LIN {X 0,Y 135.979,Z 327.541,A -85,B 0,C 180,E1 -24797.792,E2 -24797.792} C_VEL
LIN {X 0,Y 136.06,Z 327.536,A -85,B 0,C 180,E1 -24801.701,E2 -24801.701} C_VEL
LIN {X 0,Y 136.276,Z 327.502,A -85,B 0,C 180,E1 -24805.604,E2 -24805.604} C_VEL
LIN {X 0,Y 136.39,Z 327.497,A -85,B 0,C 180,E1 -24808.988,E2 -24808.988} C_VEL
LIN {X 0,Y 135.911,Z 327.699,A -85,B 0,C 180,E1 -24810.982,E2 -24810.982} C_VEL
LIN {X 0,Y 135.083,Z 332.653,A -85,B 0,C 180,E1 -24817.037,E2 -24817.037} C_VEL
LIN {X 0,Y 134.416,Z 337.78,A -85,B 0,C 180,E1 -24823.292,E2 -24823.292} C_VEL
LIN {X 0,Y 135.153,Z 344.313,A -85,B 0,C 180,E1 -24831.118,E2 -24831.118} C_VEL
LIN {X 0,Y 135.675,Z 345.242,A -85,B 0,C 180,E1 -24832.189,E2 -24832.189} C_VEL
LIN {X 0,Y 136.863,Z 354.975,A -85,B 0,C 180,E1 -24833.739,E2 -24833.739} C_VEL
LIN {X 0,Y 136.657,Z 365.063,A -85,B 0,C 180,E1 -24835.949,E2 -24835.949} C_VEL
LIN {X 0,Y 136.414,Z 375.842,A -85,B 0,C 180,E1 -24838.897,E2 -24838.897} C_VEL
LIN {X 0,Y 136.178,Z 387.286,A -85,B 0,C 180,E1 -24842.962,E2 -24842.962} C_VEL
LIN {X 0,Y 136.68,Z 397.433,A -85,B 0,C 180,E1 -24847.389,E2 -24847.389} C_VEL
LIN {X 0,Y 138.168,Z 405.675,A -85,B 0,C 180,E1 -24851.743,E2 -24851.743} C_VEL
LIN {X 0,Y 140.736,Z 412.502,A -85,B 0,C 180,E1 -24855.945,E2 -24855.945} C_VEL
LIN {X 0,Y 144.351,Z 418.057,A -85,B 0,C 180,E1 -24859.93,E2 -24859.93} C_VEL
LIN {X 0,Y 148.855,Z 422.491,A -85,B 0,C 180,E1 -24863.664,E2 -24863.664} C_VEL
LIN {X 0,Y 154.201,Z 425.904,A -85,B 0,C 180,E1 -24867.118,E2 -24867.118} C_VEL
LIN {X 0,Y 158.207,Z 427.606,A -85,B 0,C 180,E1 -24869.255,E2 -24869.255} C_VEL
LIN {X 0,Y 162.506,Z 428.906,A -85,B 0,C 180,E1 -24871.267,E2 -24871.267} C_VEL
LIN {X 0,Y 170.287,Z 430.119,A -85,B 0,C 180,E1 -24874.368,E2 -24874.368} C_VEL
LIN {X 0,Y 176.196,Z 430.401,A -85,B 0,C 180,E1 -24876.752,E2 -24876.752} C_VEL
LIN {X 0,Y 178.308,Z 430.889,A -85,B 0,C 180,E1 -24879.1,E2 -24879.1} C_VEL
LIN {X 0,Y 179.822,Z 431.717,A -85,B 0,C 180,E1 -24882.048,E2 -24882.048} C_VEL
LIN {X 0,Y 179.602,Z 432.393,A -85,B 0,C 180,E1 -24883.62,E2 -24883.62} C_VEL
LIN {X 0,Y 177.592,Z 433.122,A -85,B 0,C 180,E1 -24884.575,E2 -24884.575} C_VEL
LIN {X 0,Y 167.705,Z 435.389,A -85,B 0,C 180,E1 -24887.893,E2 -24887.893} C_VEL
LIN {X 0,Y 158.877,Z 436.572,A -85,B 0,C 180,E1 -24891.735,E2 -24891.735} C_VEL
LIN {X 0,Y 151.362,Z 436.718,A -85,B 0,C 180,E1 -24896.139,E2 -24896.139} C_VEL
LIN {X 0,Y 145.311,Z 435.829,A -85,B 0,C 180,E1 -24901.076,E2 -24901.076} C_VEL
LIN {X 0,Y 141.019,Z 433.963,A -85,B 0,C 180,E1 -24906.503,E2 -24906.503} C_VEL
LIN {X 0,Y 138.563,Z 431.066,A -85,B 0,C 180,E1 -24912.282,E2 -24912.282} C_VEL
LIN {X 0,Y 138.068,Z 427.043,A -85,B 0,C 180,E1 -24918.252,E2 -24918.252} C_VEL
LIN {X 0,Y 139.403,Z 421.603,A -85,B 0,C 180,E1 -24924.213,E2 -24924.213} C_VEL
LIN {X 0,Y 140.672,Z 417.257,A -85,B 0,C 180,E1 -24927.791,E2 -24927.791} C_VEL
LIN {X 0,Y 142.352,Z 411.13,A -85,B 0,C 180,E1 -24931.702,E2 -24931.702} C_VEL
LIN {X 0,Y 144.37,Z 407.507,A -85,B 0,C 180,E1 -24933.874,E2 -24933.874} C_VEL
LIN {X 0,Y 141.887,Z 414.835,A -85,B 0,C 180,E1 -24937.82,E2 -24937.82} C_VEL
LIN {X 0,Y 140.373,Z 420.237,A -85,B 0,C 180,E1 -24941.553,E2 -24941.553} C_VEL
LIN {X 0,Y 139.886,Z 425.653,A -85,B 0,C 180,E1 -24946.414,E2 -24946.414} C_VEL
LIN {X 0,Y 141.433,Z 430.393,A -85,B 0,C 180,E1 -24951.881,E2 -24951.881} C_VEL
LIN {X 0,Y 144.15,Z 433.099,A -85,B 0,C 180,E1 -24956.027,E2 -24956.027} C_VEL
LIN {X 0,Y 146.64,Z 434.437,A -85,B 0,C 180,E1 -24958.638,E2 -24958.638} C_VEL
LIN {X 0,Y 149.609,Z 435.401,A -85,B 0,C 180,E1 -24961.114,E2 -24961.114} C_VEL
LIN {X 0,Y 153.036,Z 435.977,A -85,B 0,C 180,E1 -24963.442,E2 -24963.442} C_VEL
LIN {X 0,Y 156.96,Z 436.164,A -85,B 0,C 180,E1 -24965.598,E2 -24965.598} C_VEL
LIN {X 0,Y 161.236,Z 435.912,A -85,B 0,C 180,E1 -24967.607,E2 -24967.607} C_VEL
LIN {X 0,Y 165.846,Z 435.255,A -85,B 0,C 180,E1 -24969.468,E2 -24969.468} C_VEL
LIN {X 0,Y 170.838,Z 434.17,A -85,B 0,C 180,E1 -24971.164,E2 -24971.164} C_VEL
LIN {X 0,Y 178.821,Z 431.68,A -85,B 0,C 180,E1 -24973.455,E2 -24973.455} C_VEL
LIN {X 0,Y 183.487,Z 429.679,A -85,B 0,C 180,E1 -24974.829,E2 -24974.829} C_VEL
LIN {X 0,Y 182.659,Z 429.091,A -85,B 0,C 180,E1 -24976.974,E2 -24976.974} C_VEL
LIN {X 0,Y 181.359,Z 428.903,A -85,B 0,C 180,E1 -24978.79,E2 -24978.79} C_VEL
LIN {X 0,Y 178.916,Z 428.831,A -85,B 0,C 180,E1 -24981.058,E2 -24981.058} C_VEL
LIN {X 0,Y 176.005,Z 428.924,A -85,B 0,C 180,E1 -24983.201,E2 -24983.201} C_VEL
LIN {X 0,Y 172.17,Z 428.982,A -85,B 0,C 180,E1 -24985.143,E2 -24985.143} C_VEL
LIN {X 0,Y 167.361,Z 428.804,A -85,B 0,C 180,E1 -24986.91,E2 -24986.91} C_VEL
LIN {X 0,Y 162.753,Z 428.071,A -85,B 0,C 180,E1 -24988.786,E2 -24988.786} C_VEL
LIN {X 0,Y 158.415,Z 426.792,A -85,B 0,C 180,E1 -24990.787,E2 -24990.787} C_VEL
LIN {X 0,Y 152.538,Z 423.815,A -85,B 0,C 180,E1 -24994.039,E2 -24994.039} C_VEL
LIN {X 0,Y 150.428,Z 422.316,A -85,B 0,C 180,E1 -24995.385,E2 -24995.385} C_VEL
LIN {X 0,Y 147.381,Z 420.031,A -85,B 0,C 180,E1 -24997.089,E2 -24997.089} C_VEL
LIN {X 0,Y 143.823,Z 417.312,A -85,B 0,C 180,E1 -24998.608,E2 -24998.608} C_VEL
LIN {X 0,Y 137.001,Z 410.655,A -85,B 0,C 180,E1 -25001.573,E2 -25001.573} C_VEL
LIN {X 0,Y 134.667,Z 406.952,A -85,B 0,C 180,E1 -25003.278,E2 -25003.278} C_VEL
LIN {X 0,Y 134.183,Z 405.673,A -85,B 0,C 180,E1 -25003.906,E2 -25003.906} C_VEL
LIN {X 0,Y 132.351,Z 397.688,A -85,B 0,C 180,E1 -25007.733,E2 -25007.733} C_VEL
LIN {X 0,Y 131.623,Z 388.06,A -85,B 0,C 180,E1 -25011.552,E2 -25011.552} C_VEL
LIN {X 0,Y 131.713,Z 378.411,A -85,B 0,C 180,E1 -25014.638,E2 -25014.638} C_VEL
LIN {X 0,Y 132.18,Z 369.208,A -85,B 0,C 180,E1 -25016.948,E2 -25016.948} C_VEL
LIN {X 0,Y 132.386,Z 364.406,A -85,B 0,C 180,E1 -25017.904,E2 -25017.904} C_VEL
LIN {X 0,Y 127.928,Z 339.902,A -85,B 0,C 180,E1 -25036.759,E2 -25036.759} C_VEL
LIN {X 0,Y 128.249,Z 331.535,A -85,B 0,C 180,E1 -25043.405,E2 -25043.405} C_VEL
LIN {X 0,Y 128.472,Z 328.482,A -85,B 0,C 180,E1 -25045.948,E2 -25045.948} C_VEL
LIN {X 0,Y 128.911,Z 328.428,A -85,B 0,C 180,E1 -25049.379,E2 -25049.379} C_VEL
LIN {X 0,Y 128.987,Z 328.412,A -85,B 0,C 180,E1 -25055.185,E2 -25055.185} C_VEL
LIN {X 0,Y 128.917,Z 328.425,A -85,B 0,C 180,E1 -25060.852,E2 -25060.852} C_VEL
LIN {X 0,Y 128.905,Z 328.426,A -85,B 0,C 180,E1 -25065.129,E2 -25065.129} C_VEL
LIN {X 0,Y 128.928,Z 328.422,A -85,B 0,C 180,E1 -25069.736,E2 -25069.736} C_VEL
LIN {X 0,Y 128.973,Z 328.42,A -85,B 0,C 180,E1 -25074.816,E2 -25074.816} C_VEL
LIN {X 0,Y 129.008,Z 328.409,A -85,B 0,C 180,E1 -25080.64,E2 -25080.64} C_VEL
LIN {X 0,Y 129.022,Z 328.413,A -85,B 0,C 180,E1 -25084.166,E2 -25084.166} C_VEL
LIN {X 0,Y 129.099,Z 328.399,A -85,B 0,C 180,E1 -25087.726,E2 -25087.726} C_VEL
LIN {X 0,Y 129.147,Z 328.397,A -85,B 0,C 180,E1 -25090.943,E2 -25090.943} C_VEL
LIN {X 0,Y 129.38,Z 328.362,A -85,B 0,C 180,E1 -25097.875,E2 -25097.875} C_VEL
LIN {X 0,Y 129.461,Z 328.359,A -85,B 0,C 180,E1 -25100.627,E2 -25100.627} C_VEL
LIN {X 0,Y 130.057,Z 328.286,A -85,B 0,C 180,E1 -25110,E2 -25110} C_VEL
LIN {X 0,Y 129.461,Z 328.359,A -85,B 0,C 180,E1 -25119.373,E2 -25119.373} C_VEL
LIN {X 0,Y 129.336,Z 328.367,A -85,B 0,C 180,E1 -25122.554,E2 -25122.554} C_VEL
LIN {X 0,Y 129.17,Z 328.394,A -85,B 0,C 180,E1 -25129.054,E2 -25129.054} C_VEL
LIN {X 0,Y 129.127,Z 328.396,A -85,B 0,C 180,E1 -25132.395,E2 -25132.395} C_VEL
LIN {X 0,Y 129.028,Z 328.407,A -85,B 0,C 180,E1 -25139.376,E2 -25139.376} C_VEL
LIN {X 0,Y 128.973,Z 328.42,A -85,B 0,C 180,E1 -25145.184,E2 -25145.184} C_VEL
LIN {X 0,Y 128.917,Z 328.424,A -85,B 0,C 180,E1 -25150.858,E2 -25150.858} C_VEL
LIN {X 0,Y 128.905,Z 328.425,A -85,B 0,C 180,E1 -25155.135,E2 -25155.135} C_VEL
LIN {X 0,Y 128.942,Z 328.422,A -85,B 0,C 180,E1 -25159.736,E2 -25159.736} C_VEL
LIN {X 0,Y 129.139,Z 328.394,A -85,B 0,C 180,E1 -25164.72,E2 -25164.72} C_VEL
LIN {X 0,Y 129.235,Z 328.383,A -85,B 0,C 180,E1 -25167.061,E2 -25167.061} C_VEL
LIN {X 0,Y 128.692,Z 328.577,A -85,B 0,C 180,E1 -25171.572,E2 -25171.572} C_VEL
LIN {X 0,Y 127.933,Z 333.105,A -85,B 0,C 180,E1 -25177.389,E2 -25177.389} C_VEL
LIN {X 0,Y 127.276,Z 338.27,A -85,B 0,C 180,E1 -25183.977,E2 -25183.977} C_VEL
LIN {X 0,Y 128.495,Z 344.938,A -85,B 0,C 180,E1 -25192.351,E2 -25192.351} C_VEL
LIN {X 0,Y 128.938,Z 345.731,A -85,B 0,C 180,E1 -25193.148,E2 -25193.148} C_VEL
LIN {X 0,Y 130.047,Z 354.44,A -85,B 0,C 180,E1 -25194.577,E2 -25194.577} C_VEL
LIN {X 0,Y 129.881,Z 364.497,A -85,B 0,C 180,E1 -25196.902,E2 -25196.902} C_VEL
LIN {X 0,Y 129.768,Z 374.013,A -85,B 0,C 180,E1 -25199.616,E2 -25199.616} C_VEL
LIN {X 0,Y 129.529,Z 383.947,A -85,B 0,C 180,E1 -25203.114,E2 -25203.114} C_VEL
LIN {X 0,Y 129.858,Z 393.128,A -85,B 0,C 180,E1 -25206.998,E2 -25206.998} C_VEL
LIN {X 0,Y 131.157,Z 402.14,A -85,B 0,C 180,E1 -25211.596,E2 -25211.596} C_VEL
LIN {X 0,Y 133.538,Z 409.687,A -85,B 0,C 180,E1 -25216.044,E2 -25216.044} C_VEL
LIN {X 0,Y 137.758,Z 416.78,A -85,B 0,C 180,E1 -25220.927,E2 -25220.927} C_VEL
LIN {X 0,Y 142.391,Z 421.671,A -85,B 0,C 180,E1 -25224.809,E2 -25224.809} C_VEL
LIN {X 0,Y 147.893,Z 425.491,A -85,B 0,C 180,E1 -25228.377,E2 -25228.377} C_VEL
LIN {X 0,Y 152.021,Z 427.502,A -85,B 0,C 180,E1 -25230.57,E2 -25230.57} C_VEL
LIN {X 0,Y 156.454,Z 429.083,A -85,B 0,C 180,E1 -25232.622,E2 -25232.622} C_VEL
LIN {X 0,Y 164.94,Z 430.874,A -85,B 0,C 180,E1 -25235.945,E2 -25235.945} C_VEL
LIN {X 0,Y 166.079,Z 431.002,A -85,B 0,C 180,E1 -25236.334,E2 -25236.334} C_VEL
LIN {X 0,Y 170.321,Z 431.518,A -85,B 0,C 180,E1 -25238.243,E2 -25238.243} C_VEL
LIN {X 0,Y 172.095,Z 432.303,A -85,B 0,C 180,E1 -25240.802,E2 -25240.802} C_VEL
LIN {X 0,Y 172.594,Z 433.048,A -85,B 0,C 180,E1 -25242.865,E2 -25242.865} C_VEL
LIN {X 0,Y 162.533,Z 434.785,A -85,B 0,C 180,E1 -25246.223,E2 -25246.223} C_VEL
LIN {X 0,Y 153.433,Z 435.466,A -85,B 0,C 180,E1 -25250.113,E2 -25250.113} C_VEL
LIN {X 0,Y 145.65,Z 435.17,A -85,B 0,C 180,E1 -25254.617,E2 -25254.617} C_VEL
LIN {X 0,Y 139.369,Z 433.885,A -85,B 0,C 180,E1 -25259.717,E2 -25259.717} C_VEL
LIN {X 0,Y 134.86,Z 431.648,A -85,B 0,C 180,E1 -25265.36,E2 -25265.36} C_VEL
LIN {X 0,Y 132.281,Z 428.393,A -85,B 0,C 180,E1 -25271.411,E2 -25271.411} C_VEL
LIN {X 0,Y 131.754,Z 424.034,A -85,B 0,C 180,E1 -25277.68,E2 -25277.68} C_VEL
LIN {X 0,Y 133.18,Z 418.274,A -85,B 0,C 180,E1 -25283.942,E2 -25283.942} C_VEL
LIN {X 0,Y 134.503,Z 413.642,A -85,B 0,C 180,E1 -25287.69,E2 -25287.69} C_VEL
LIN {X 0,Y 136.475,Z 406.993,A -85,B 0,C 180,E1 -25291.898,E2 -25291.898} C_VEL
LIN {X 0,Y 138.897,Z 403.116,A -85,B 0,C 180,E1 -25294.28,E2 -25294.28} C_VEL
LIN {X 0,Y 136.176,Z 410.644,A -85,B 0,C 180,E1 -25298.15,E2 -25298.15} C_VEL
LIN {X 0,Y 134.564,Z 416.341,A -85,B 0,C 180,E1 -25302.059,E2 -25302.059} C_VEL
LIN {X 0,Y 133.906,Z 421.325,A -85,B 0,C 180,E1 -25306.284,E2 -25306.284} C_VEL
LIN {X 0,Y 134.814,Z 426.291,A -85,B 0,C 180,E1 -25311.403,E2 -25311.403} C_VEL
LIN {X 0,Y 136.199,Z 428.656,A -85,B 0,C 180,E1 -25314.381,E2 -25314.381} C_VEL
LIN {X 0,Y 138.201,Z 430.639,A -85,B 0,C 180,E1 -25317.238,E2 -25317.238} C_VEL
LIN {X 0,Y 140.76,Z 432.23,A -85,B 0,C 180,E1 -25319.953,E2 -25319.953} C_VEL
LIN {X 0,Y 147.323,Z 434.326,A -85,B 0,C 180,E1 -25324.922,E2 -25324.922} C_VEL
LIN {X 0,Y 151.341,Z 434.852,A -85,B 0,C 180,E1 -25327.135,E2 -25327.135} C_VEL
LIN {X 0,Y 155.732,Z 434.988,A -85,B 0,C 180,E1 -25329.184,E2 -25329.184} C_VEL
LIN {X 0,Y 160.443,Z 434.685,A -85,B 0,C 180,E1 -25331.076,E2 -25331.076} C_VEL
LIN {X 0,Y 165.554,Z 433.973,A -85,B 0,C 180,E1 -25332.783,E2 -25332.783} C_VEL
LIN {X 0,Y 170.948,Z 432.822,A -85,B 0,C 180,E1 -25334.339,E2 -25334.339} C_VEL
LIN {X 0,Y 176.254,Z 431.265,A -85,B 0,C 180,E1 -25335.868,E2 -25335.868} C_VEL
LIN {X 0,Y 175.546,Z 430.96,A -85,B 0,C 180,E1 -25337.106,E2 -25337.106} C_VEL
LIN {X 0,Y 173.23,Z 430.557,A -85,B 0,C 180,E1 -25339.521,E2 -25339.521} C_VEL
LIN {X 0,Y 170.342,Z 430.266,A -85,B 0,C 180,E1 -25341.763,E2 -25341.763} C_VEL
LIN {X 0,Y 166.388,Z 429.931,A -85,B 0,C 180,E1 -25343.744,E2 -25343.744} C_VEL
LIN {X 0,Y 161.432,Z 429.339,A -85,B 0,C 180,E1 -25345.527,E2 -25345.527} C_VEL
LIN {X 0,Y 156.681,Z 428.21,A -85,B 0,C 180,E1 -25347.431,E2 -25347.431} C_VEL
LIN {X 0,Y 150.121,Z 425.546,A -85,B 0,C 180,E1 -25350.553,E2 -25350.553} C_VEL
LIN {X 0,Y 144.328,Z 421.541,A -85,B 0,C 180,E1 -25354.004,E2 -25354.004} C_VEL
LIN {X 0,Y 139.447,Z 416.299,A -85,B 0,C 180,E1 -25357.787,E2 -25357.787} C_VEL
LIN {X 0,Y 136.156,Z 410.722,A -85,B 0,C 180,E1 -25361.175,E2 -25361.175} C_VEL
LIN {X 0,Y 134.183,Z 405.673,A -85,B 0,C 180,E1 -25363.906,E2 -25363.906} C_VEL
LIN {X 0,Y 132.597,Z 401.763,A -85,B 0,C 180,E1 -25365.657,E2 -25365.657} C_VEL
LIN {X 0,Y 129.033,Z 394.378,A -85,B 0,C 180,E1 -25368.074,E2 -25368.074} C_VEL
LIN {X 0,Y 126.08,Z 386.22,A -85,B 0,C 180,E1 -25370.333,E2 -25370.333} C_VEL
LIN {X 0,Y 125.532,Z 381.233,A -85,B 0,C 180,E1 -25371.814,E2 -25371.814} C_VEL
LIN {X 0,Y 125.79,Z 372.273,A -85,B 0,C 180,E1 -25374.385,E2 -25374.385} C_VEL
LIN {X 0,Y 126.176,Z 365.058,A -85,B 0,C 180,E1 -25376.103,E2 -25376.103} C_VEL
LIN {X 0,Y 120.807,Z 340.148,A -85,B 0,C 180,E1 -25396.037,E2 -25396.037} C_VEL
LIN {X 0,Y 121.1,Z 332.348,A -85,B 0,C 180,E1 -25402.529,E2 -25402.529} C_VEL
LIN {X 0,Y 121.308,Z 329.374,A -85,B 0,C 180,E1 -25405.06,E2 -25405.06} C_VEL
LIN {X 0,Y 121.862,Z 329.305,A -85,B 0,C 180,E1 -25410.108,E2 -25410.108} C_VEL
LIN {X 0,Y 121.899,Z 329.298,A -85,B 0,C 180,E1 -25416.18,E2 -25416.18} C_VEL
LIN {X 0,Y 121.857,Z 329.301,A -85,B 0,C 180,E1 -25421.43,E2 -25421.43} C_VEL
LIN {X 0,Y 121.857,Z 329.306,A -85,B 0,C 180,E1 -25428.563,E2 -25428.563} C_VEL
LIN {X 0,Y 121.925,Z 329.298,A -85,B 0,C 180,E1 -25434.801,E2 -25434.801} C_VEL
LIN {X 0,Y 121.92,Z 329.291,A -85,B 0,C 180,E1 -25439.834,E2 -25439.834} C_VEL
LIN {X 0,Y 121.975,Z 329.29,A -85,B 0,C 180,E1 -25446.213,E2 -25446.213} C_VEL
LIN {X 0,Y 122.038,Z 329.278,A -85,B 0,C 180,E1 -25449.786,E2 -25449.786} C_VEL
LIN {X 0,Y 122.231,Z 329.252,A -85,B 0,C 180,E1 -25456.703,E2 -25456.703} C_VEL
LIN {X 0,Y 122.398,Z 329.238,A -85,B 0,C 180,E1 -25460.081,E2 -25460.081} C_VEL
LIN {X 0,Y 122.551,Z 329.215,A -85,B 0,C 180,E1 -25466.712,E2 -25466.712} C_VEL
LIN {X 0,Y 123.011,Z 329.163,A -85,B 0,C 180,E1 -25470,E2 -25470} C_VEL
LIN {X 0,Y 122.4,Z 329.237,A -85,B 0,C 180,E1 -25476.594,E2 -25476.594} C_VEL
LIN {X 0,Y 122.398,Z 329.238,A -85,B 0,C 180,E1 -25479.919,E2 -25479.919} C_VEL
LIN {X 0,Y 122.232,Z 329.252,A -85,B 0,C 180,E1 -25483.296,E2 -25483.296} C_VEL
LIN {X 0,Y 122.06,Z 329.276,A -85,B 0,C 180,E1 -25490.211,E2 -25490.211} C_VEL
LIN {X 0,Y 121.988,Z 329.289,A -85,B 0,C 180,E1 -25493.784,E2 -25493.784} C_VEL
LIN {X 0,Y 121.933,Z 329.289,A -85,B 0,C 180,E1 -25500.176,E2 -25500.176} C_VEL
LIN {X 0,Y 121.889,Z 329.3,A -85,B 0,C 180,E1 -25506.183,E2 -25506.183} C_VEL
LIN {X 0,Y 121.857,Z 329.306,A -85,B 0,C 180,E1 -25511.437,E2 -25511.437} C_VEL
LIN {X 0,Y 121.864,Z 329.3,A -85,B 0,C 180,E1 -25518.566,E2 -25518.566} C_VEL
LIN {X 0,Y 122.094,Z 329.27,A -85,B 0,C 180,E1 -25524.862,E2 -25524.862} C_VEL
LIN {X 0,Y 121.889,Z 329.304,A -85,B 0,C 180,E1 -25529.87,E2 -25529.87} C_VEL
LIN {X 0,Y 121.452,Z 329.586,A -85,B 0,C 180,E1 -25532.429,E2 -25532.429} C_VEL
LIN {X 0,Y 120.678,Z 334.258,A -85,B 0,C 180,E1 -25538.718,E2 -25538.718} C_VEL
LIN {X 0,Y 120.883,Z 343.579,A -85,B 0,C 180,E1 -25551.251,E2 -25551.251} C_VEL
LIN {X 0,Y 122.276,Z 345.925,A -85,B 0,C 180,E1 -25554.232,E2 -25554.232} C_VEL
LIN {X 0,Y 123.425,Z 355.351,A -85,B 0,C 180,E1 -25555.923,E2 -25555.923} C_VEL
LIN {X 0,Y 123.225,Z 368.066,A -85,B 0,C 180,E1 -25559.187,E2 -25559.187} C_VEL
LIN {X 0,Y 122.989,Z 378.06,A -85,B 0,C 180,E1 -25562.461,E2 -25562.461} C_VEL
LIN {X 0,Y 123.176,Z 388.165,A -85,B 0,C 180,E1 -25566.557,E2 -25566.557} C_VEL
LIN {X 0,Y 124.25,Z 398.142,A -85,B 0,C 180,E1 -25571.423,E2 -25571.423} C_VEL
LIN {X 0,Y 126.499,Z 406.389,A -85,B 0,C 180,E1 -25576.132,E2 -25576.132} C_VEL
LIN {X 0,Y 130.564,Z 414.29,A -85,B 0,C 180,E1 -25581.309,E2 -25581.309} C_VEL
LIN {X 0,Y 134.328,Z 418.931,A -85,B 0,C 180,E1 -25584.747,E2 -25584.747} C_VEL
LIN {X 0,Y 139.699,Z 423.542,A -85,B 0,C 180,E1 -25588.554,E2 -25588.554} C_VEL
LIN {X 0,Y 145.932,Z 427.144,A -85,B 0,C 180,E1 -25591.993,E2 -25591.993} C_VEL
LIN {X 0,Y 155.328,Z 430.504,A -85,B 0,C 180,E1 -25596.033,E2 -25596.033} C_VEL
LIN {X 0,Y 160.37,Z 431.552,A -85,B 0,C 180,E1 -25597.849,E2 -25597.849} C_VEL
LIN {X 0,Y 163.896,Z 432.229,A -85,B 0,C 180,E1 -25599.479,E2 -25599.479} C_VEL
LIN {X 0,Y 165.011,Z 433.181,A -85,B 0,C 180,E1 -25601.975,E2 -25601.975} C_VEL
LIN {X 0,Y 157.538,Z 433.935,A -85,B 0,C 180,E1 -25604.456,E2 -25604.456} C_VEL
LIN {X 0,Y 148.162,Z 434.139,A -85,B 0,C 180,E1 -25608.388,E2 -25608.388} C_VEL
LIN {X 0,Y 140.086,Z 433.385,A -85,B 0,C 180,E1 -25612.984,E2 -25612.984} C_VEL
LIN {X 0,Y 133.563,Z 431.721,A -85,B 0,C 180,E1 -25618.251,E2 -25618.251} C_VEL
LIN {X 0,Y 128.849,Z 429.116,A -85,B 0,C 180,E1 -25624.128,E2 -25624.128} C_VEL
LIN {X 0,Y 125.85,Z 424.735,A -85,B 0,C 180,E1 -25631.698,E2 -25631.698} C_VEL
LIN {X 0,Y 125.791,Z 419.455,A -85,B 0,C 180,E1 -25638.723,E2 -25638.723} C_VEL
LIN {X 0,Y 127.211,Z 414.357,A -85,B 0,C 180,E1 -25643.992,E2 -25643.992} C_VEL
LIN {X 0,Y 128.499,Z 409.542,A -85,B 0,C 180,E1 -25647.757,E2 -25647.757} C_VEL
LIN {X 0,Y 130.924,Z 402.291,A -85,B 0,C 180,E1 -25652.307,E2 -25652.307} C_VEL
LIN {X 0,Y 133.56,Z 398.564,A -85,B 0,C 180,E1 -25654.716,E2 -25654.716} C_VEL
LIN {X 0,Y 130.81,Z 405.888,A -85,B 0,C 180,E1 -25658.416,E2 -25658.416} C_VEL
LIN {X 0,Y 128.929,Z 412.216,A -85,B 0,C 180,E1 -25662.594,E2 -25662.594} C_VEL
LIN {X 0,Y 128.158,Z 418.801,A -85,B 0,C 180,E1 -25668.165,E2 -25668.165} C_VEL
LIN {X 0,Y 129.01,Z 422.93,A -85,B 0,C 180,E1 -25672.417,E2 -25672.417} C_VEL
LIN {X 0,Y 131.341,Z 426.786,A -85,B 0,C 180,E1 -25677.054,E2 -25677.054} C_VEL
LIN {X 0,Y 135.044,Z 429.761,A -85,B 0,C 180,E1 -25681.361,E2 -25681.361} C_VEL
LIN {X 0,Y 138.185,Z 431.276,A -85,B 0,C 180,E1 -25684.018,E2 -25684.018} C_VEL
LIN {X 0,Y 141.777,Z 432.39,A -85,B 0,C 180,E1 -25686.502,E2 -25686.502} C_VEL
LIN {X 0,Y 145.893,Z 433.221,A -85,B 0,C 180,E1 -25688.773,E2 -25688.773} C_VEL
LIN {X 0,Y 150.387,Z 433.687,A -85,B 0,C 180,E1 -25690.864,E2 -25690.864} C_VEL
LIN {X 0,Y 155.207,Z 433.782,A -85,B 0,C 180,E1 -25692.783,E2 -25692.783} C_VEL
LIN {X 0,Y 160.428,Z 433.469,A -85,B 0,C 180,E1 -25694.502,E2 -25694.502} C_VEL
LIN {X 0,Y 167.727,Z 432.402,A -85,B 0,C 180,E1 -25696.565,E2 -25696.565} C_VEL
LIN {X 0,Y 167.485,Z 431.957,A -85,B 0,C 180,E1 -25697.822,E2 -25697.822} C_VEL
LIN {X 0,Y 164.707,Z 431.269,A -85,B 0,C 180,E1 -25700.201,E2 -25700.201} C_VEL
LIN {X 0,Y 160.685,Z 430.594,A -85,B 0,C 180,E1 -25702.238,E2 -25702.238} C_VEL
LIN {X 0,Y 155.588,Z 429.599,A -85,B 0,C 180,E1 -25704.036,E2 -25704.036} C_VEL
LIN {X 0,Y 148.408,Z 427.12,A -85,B 0,C 180,E1 -25706.999,E2 -25706.999} C_VEL
LIN {X 0,Y 141.923,Z 423.402,A -85,B 0,C 180,E1 -25710.313,E2 -25710.313} C_VEL
LIN {X 0,Y 136.297,Z 418.421,A -85,B 0,C 180,E1 -25714.001,E2 -25714.001} C_VEL
LIN {X 0,Y 131.672,Z 411.986,A -85,B 0,C 180,E1 -25718.057,E2 -25718.057} C_VEL
LIN {X 0,Y 128.127,Z 403.878,A -85,B 0,C 180,E1 -25722.504,E2 -25722.504} C_VEL
LIN {X 0,Y 126.334,Z 395.716,A -85,B 0,C 180,E1 -25726.32,E2 -25726.32} C_VEL
LIN {X 0,Y 125.556,Z 386.77,A -85,B 0,C 180,E1 -25729.922,E2 -25729.922} C_VEL
LIN {X 0,Y 125.532,Z 381.233,A -85,B 0,C 180,E1 -25731.814,E2 -25731.814} C_VEL
LIN {X 0,Y 124.969,Z 377.479,A -85,B 0,C 180,E1 -25732.765,E2 -25732.765} C_VEL
LIN {X 0,Y 123.008,Z 371.864,A -85,B 0,C 180,E1 -25733.566,E2 -25733.566} C_VEL
LIN {X 0,Y 120.22,Z 365.879,A -85,B 0,C 180,E1 -25734.727,E2 -25734.727} C_VEL
LIN {X 0,Y 119.024,Z 363.495,A -85,B 0,C 180,E1 -25735.761,E2 -25735.761} C_VEL
LIN {X 0,Y 118.831,Z 363.119,A -85,B 0,C 180,E1 -25736.022,E2 -25736.022} C_VEL
LIN {X 0,Y 113.76,Z 339.277,A -85,B 0,C 180,E1 -25756.136,E2 -25756.136} C_VEL
LIN {X 0,Y 114.025,Z 332.111,A -85,B 0,C 180,E1 -25762.402,E2 -25762.402} C_VEL
LIN {X 0,Y 114.122,Z 330.268,A -85,B 0,C 180,E1 -25764.19,E2 -25764.19} C_VEL
LIN {X 0,Y 114.702,Z 330.198,A -85,B 0,C 180,E1 -25769.346,E2 -25769.346} C_VEL
LIN {X 0,Y 114.818,Z 330.176,A -85,B 0,C 180,E1 -25773.422,E2 -25773.422} C_VEL
LIN {X 0,Y 114.783,Z 330.187,A -85,B 0,C 180,E1 -25777.749,E2 -25777.749} C_VEL
LIN {X 0,Y 114.771,Z 330.182,A -85,B 0,C 180,E1 -25782.708,E2 -25782.708} C_VEL
LIN {X 0,Y 114.779,Z 330.187,A -85,B 0,C 180,E1 -25787.659,E2 -25787.659} C_VEL
LIN {X 0,Y 114.788,Z 330.181,A -85,B 0,C 180,E1 -25792.736,E2 -25792.736} C_VEL
LIN {X 0,Y 114.854,Z 330.172,A -85,B 0,C 180,E1 -25798.935,E2 -25798.935} C_VEL
LIN {X 0,Y 114.939,Z 330.165,A -85,B 0,C 180,E1 -25806.504,E2 -25806.504} C_VEL
LIN {X 0,Y 115.004,Z 330.16,A -85,B 0,C 180,E1 -25812.208,E2 -25812.208} C_VEL
LIN {X 0,Y 115.239,Z 330.122,A -85,B 0,C 180,E1 -25817.34,E2 -25817.34} C_VEL
LIN {X 0,Y 115.344,Z 330.116,A -85,B 0,C 180,E1 -25823,E2 -25823} C_VEL
LIN {X 0,Y 115.963,Z 330.041,A -85,B 0,C 180,E1 -25830,E2 -25830} C_VEL
LIN {X 0,Y 115.344,Z 330.116,A -85,B 0,C 180,E1 -25837,E2 -25837} C_VEL
LIN {X 0,Y 115.239,Z 330.122,A -85,B 0,C 180,E1 -25842.66,E2 -25842.66} C_VEL
LIN {X 0,Y 115.017,Z 330.158,A -85,B 0,C 180,E1 -25847.79,E2 -25847.79} C_VEL
LIN {X 0,Y 114.957,Z 330.163,A -85,B 0,C 180,E1 -25853.516,E2 -25853.516} C_VEL
LIN {X 0,Y 114.859,Z 330.172,A -85,B 0,C 180,E1 -25861.07,E2 -25861.07} C_VEL
LIN {X 0,Y 114.777,Z 330.181,A -85,B 0,C 180,E1 -25867.757,E2 -25867.757} C_VEL
LIN {X 0,Y 114.772,Z 330.189,A -85,B 0,C 180,E1 -25872.716,E2 -25872.716} C_VEL
LIN {X 0,Y 114.784,Z 330.181,A -85,B 0,C 180,E1 -25877.668,E2 -25877.668} C_VEL
LIN {X 0,Y 114.901,Z 330.172,A -85,B 0,C 180,E1 -25882.67,E2 -25882.67} C_VEL
LIN {X 0,Y 114.904,Z 330.172,A -85,B 0,C 180,E1 -25888.904,E2 -25888.904} C_VEL
LIN {X 0,Y 114.257,Z 330.334,A -85,B 0,C 180,E1 -25893.028,E2 -25893.028} C_VEL
LIN {X 0,Y 113.639,Z 333.95,A -85,B 0,C 180,E1 -25898.224,E2 -25898.224} C_VEL
LIN {X 0,Y 114.327,Z 344.329,A -85,B 0,C 180,E1 -25912.943,E2 -25912.943} C_VEL
LIN {X 0,Y 115.715,Z 346.303,A -85,B 0,C 180,E1 -25915.541,E2 -25915.541} C_VEL
LIN {X 0,Y 116.761,Z 354.204,A -85,B 0,C 180,E1 -25916.986,E2 -25916.986} C_VEL
LIN {X 0,Y 116.654,Z 365.828,A -85,B 0,C 180,E1 -25920.004,E2 -25920.004} C_VEL
LIN {X 0,Y 116.537,Z 376.02,A -85,B 0,C 180,E1 -25923.462,E2 -25923.462} C_VEL
LIN {X 0,Y 116.792,Z 386.477,A -85,B 0,C 180,E1 -25927.786,E2 -25927.786} C_VEL
LIN {X 0,Y 117.714,Z 395.232,A -85,B 0,C 180,E1 -25932.066,E2 -25932.066} C_VEL
LIN {X 0,Y 120.466,Z 405.263,A -85,B 0,C 180,E1 -25937.84,E2 -25937.84} C_VEL
LIN {X 0,Y 124.129,Z 412.417,A -85,B 0,C 180,E1 -25942.473,E2 -25942.473} C_VEL
LIN {X 0,Y 129.751,Z 419.22,A -85,B 0,C 180,E1 -25947.417,E2 -25947.417} C_VEL
LIN {X 0,Y 135.559,Z 423.932,A -85,B 0,C 180,E1 -25951.232,E2 -25951.232} C_VEL
LIN {X 0,Y 142.252,Z 427.678,A -85,B 0,C 180,E1 -25954.626,E2 -25954.626} C_VEL
LIN {X 0,Y 149.592,Z 430.489,A -85,B 0,C 180,E1 -25957.648,E2 -25957.648} C_VEL
LIN {X 0,Y 154.781,Z 431.839,A -85,B 0,C 180,E1 -25959.475,E2 -25959.475} C_VEL
LIN {X 0,Y 156.919,Z 432.398,A -85,B 0,C 180,E1 -25960.413,E2 -25960.413} C_VEL
LIN {X 0,Y 152.722,Z 432.835,A -85,B 0,C 180,E1 -25962.583,E2 -25962.583} C_VEL
LIN {X 0,Y 143.06,Z 432.552,A -85,B 0,C 180,E1 -25966.546,E2 -25966.546} C_VEL
LIN {X 0,Y 134.717,Z 431.364,A -85,B 0,C 180,E1 -25971.242,E2 -25971.242} C_VEL
LIN {X 0,Y 127.912,Z 429.319,A -85,B 0,C 180,E1 -25976.671,E2 -25976.671} C_VEL
LIN {X 0,Y 122.976,Z 426.351,A -85,B 0,C 180,E1 -25982.794,E2 -25982.794} C_VEL
LIN {X 0,Y 119.812,Z 421.584,A -85,B 0,C 180,E1 -25990.74,E2 -25990.74} C_VEL
LIN {X 0,Y 119.763,Z 415.948,A -85,B 0,C 180,E1 -25998.148,E2 -25998.148} C_VEL
LIN {X 0,Y 121.113,Z 410.949,A -85,B 0,C 180,E1 -26003.335,E2 -26003.335} C_VEL
LIN {X 0,Y 122.277,Z 406.806,A -85,B 0,C 180,E1 -26006.705,E2 -26006.705} C_VEL
LIN {X 0,Y 124.634,Z 399.195,A -85,B 0,C 180,E1 -26011.616,E2 -26011.616} C_VEL
LIN {X 0,Y 126.796,Z 395.558,A -85,B 0,C 180,E1 -26013.835,E2 -26013.835} C_VEL
LIN {X 0,Y 128.536,Z 393.657,A -85,B 0,C 180,E1 -26015.127,E2 -26015.127} C_VEL
LIN {X 0,Y 125.098,Z 402.518,A -85,B 0,C 180,E1 -26019.703,E2 -26019.703} C_VEL
LIN {X 0,Y 123.205,Z 409.041,A -85,B 0,C 180,E1 -26024.117,E2 -26024.117} C_VEL
LIN {X 0,Y 122.567,Z 414.17,A -85,B 0,C 180,E1 -26028.383,E2 -26028.383} C_VEL
LIN {X 0,Y 123.787,Z 420.483,A -85,B 0,C 180,E1 -26034.706,E2 -26034.706} C_VEL
LIN {X 0,Y 126.859,Z 424.771,A -85,B 0,C 180,E1 -26039.908,E2 -26039.908} C_VEL
LIN {X 0,Y 129.517,Z 426.962,A -85,B 0,C 180,E1 -26042.863,E2 -26042.863} C_VEL
LIN {X 0,Y 132.745,Z 428.771,A -85,B 0,C 180,E1 -26045.618,E2 -26045.618} C_VEL
LIN {X 0,Y 136.426,Z 430.215,A -85,B 0,C 180,E1 -26048.184,E2 -26048.184} C_VEL
LIN {X 0,Y 145.229,Z 432.072,A -85,B 0,C 180,E1 -26052.649,E2 -26052.649} C_VEL
LIN {X 0,Y 150.156,Z 432.496,A -85,B 0,C 180,E1 -26054.594,E2 -26054.594} C_VEL
LIN {X 0,Y 159.42,Z 432.357,A -85,B 0,C 180,E1 -26057.433,E2 -26057.433} C_VEL
LIN {X 0,Y 159.032,Z 431.957,A -85,B 0,C 180,E1 -26058.476,E2 -26058.476} C_VEL
LIN {X 0,Y 158.608,Z 431.793,A -85,B 0,C 180,E1 -26058.875,E2 -26058.875} C_VEL
LIN {X 0,Y 155.088,Z 430.954,A -85,B 0,C 180,E1 -26060.619,E2 -26060.619} C_VEL
LIN {X 0,Y 149.845,Z 429.555,A -85,B 0,C 180,E1 -26062.427,E2 -26062.427} C_VEL
LIN {X 0,Y 142.49,Z 426.401,A -85,B 0,C 180,E1 -26065.44,E2 -26065.44} C_VEL
LIN {X 0,Y 135.828,Z 422.14,A -85,B 0,C 180,E1 -26068.837,E2 -26068.837} C_VEL
LIN {X 0,Y 130.1,Z 416.449,A -85,B 0,C 180,E1 -26072.662,E2 -26072.662} C_VEL
LIN {X 0,Y 125.416,Z 409.436,A -85,B 0,C 180,E1 -26076.9,E2 -26076.9} C_VEL
LIN {X 0,Y 121.922,Z 400.605,A -85,B 0,C 180,E1 -26081.512,E2 -26081.512} C_VEL
LIN {X 0,Y 120.474,Z 393.561,A -85,B 0,C 180,E1 -26084.776,E2 -26084.776} C_VEL
LIN {X 0,Y 119.672,Z 384.05,A -85,B 0,C 180,E1 -26088.564,E2 -26088.564} C_VEL
LIN {X 0,Y 119.742,Z 373.448,A -85,B 0,C 180,E1 -26091.983,E2 -26091.983} C_VEL
LIN {X 0,Y 120.131,Z 365.866,A -85,B 0,C 180,E1 -26093.909,E2 -26093.909} C_VEL
LIN {X 0,Y 118.831,Z 363.119,A -85,B 0,C 180,E1 -26096.022,E2 -26096.022} C_VEL
LIN {X 0,Y 116.786,Z 360.054,A -85,B 0,C 180,E1 -26098.27,E2 -26098.27} C_VEL
LIN {X 0,Y 108.203,Z 349.832,A -85,B 0,C 180,E1 -26105.754,E2 -26105.754} C_VEL
LIN {X 0,Y 107.036,Z 346.797,A -85,B 0,C 180,E1 -26108.383,E2 -26108.383} C_VEL
LIN {X 0,Y 106.787,Z 336.183,A -85,B 0,C 180,E1 -26118.211,E2 -26118.211} C_VEL
LIN {X 0,Y 106.979,Z 331.16,A -85,B 0,C 180,E1 -26122.963,E2 -26122.963} C_VEL
LIN {X 0,Y 107.387,Z 331.109,A -85,B 0,C 180,E1 -26127.26,E2 -26127.26} C_VEL
LIN {X 0,Y 107.757,Z 331.06,A -85,B 0,C 180,E1 -26132.019,E2 -26132.019} C_VEL
LIN {X 0,Y 107.689,Z 331.07,A -85,B 0,C 180,E1 -26138.45,E2 -26138.45} C_VEL
LIN {X 0,Y 107.663,Z 331.073,A -85,B 0,C 180,E1 -26145.887,E2 -26145.887} C_VEL
LIN {X 0,Y 107.683,Z 331.064,A -85,B 0,C 180,E1 -26151.545,E2 -26151.545} C_VEL
LIN {X 0,Y 107.792,Z 331.053,A -85,B 0,C 180,E1 -26158.56,E2 -26158.56} C_VEL
LIN {X 0,Y 107.903,Z 331.04,A -85,B 0,C 180,E1 -26166.996,E2 -26166.996} C_VEL
LIN {X 0,Y 108.022,Z 331.027,A -85,B 0,C 180,E1 -26174.915,E2 -26174.915} C_VEL
LIN {X 0,Y 108.242,Z 330.998,A -85,B 0,C 180,E1 -26178.768,E2 -26178.768} C_VEL
LIN {X 0,Y 108.404,Z 330.975,A -85,B 0,C 180,E1 -26186.283,E2 -26186.283} C_VEL
LIN {X 0,Y 108.889,Z 330.922,A -85,B 0,C 180,E1 -26190,E2 -26190} C_VEL
LIN {X 0,Y 108.285,Z 330.996,A -85,B 0,C 180,E1 -26197.458,E2 -26197.458} C_VEL
LIN {X 0,Y 108.161,Z 331.004,A -85,B 0,C 180,E1 -26202.951,E2 -26202.951} C_VEL
LIN {X 0,Y 107.915,Z 331.042,A -85,B 0,C 180,E1 -26209.004,E2 -26209.004} C_VEL
LIN {X 0,Y 107.863,Z 331.048,A -85,B 0,C 180,E1 -26214.203,E2 -26214.203} C_VEL
LIN {X 0,Y 107.784,Z 331.057,A -85,B 0,C 180,E1 -26222.052,E2 -26222.052} C_VEL
LIN {X 0,Y 107.683,Z 331.064,A -85,B 0,C 180,E1 -26228.455,E2 -26228.455} C_VEL
LIN {X 0,Y 107.666,Z 331.069,A -85,B 0,C 180,E1 -26235.893,E2 -26235.893} C_VEL
LIN {X 0,Y 107.763,Z 331.061,A -85,B 0,C 180,E1 -26241.5,E2 -26241.5} C_VEL
LIN {X 0,Y 107.849,Z 331.048,A -85,B 0,C 180,E1 -26247.903,E2 -26247.903} C_VEL
LIN {X 0,Y 107.05,Z 331.193,A -85,B 0,C 180,E1 -26253.963,E2 -26253.963} C_VEL
LIN {X 0,Y 106.255,Z 335.621,A -85,B 0,C 180,E1 -26260.693,E2 -26260.693} C_VEL
LIN {X 0,Y 106.944,Z 343.371,A -85,B 0,C 180,E1 -26272.453,E2 -26272.453} C_VEL
LIN {X 0,Y 109.239,Z 346.618,A -85,B 0,C 180,E1 -26277.008,E2 -26277.008} C_VEL
LIN {X 0,Y 110.166,Z 352.741,A -85,B 0,C 180,E1 -26278.177,E2 -26278.177} C_VEL
LIN {X 0,Y 110.216,Z 364.514,A -85,B 0,C 180,E1 -26281.375,E2 -26281.375} C_VEL
LIN {X 0,Y 110.151,Z 373.78,A -85,B 0,C 180,E1 -26284.579,E2 -26284.579} C_VEL
LIN {X 0,Y 110.488,Z 384.664,A -85,B 0,C 180,E1 -26289.155,E2 -26289.155} C_VEL
LIN {X 0,Y 111.926,Z 395.177,A -85,B 0,C 180,E1 -26294.551,E2 -26294.551} C_VEL
LIN {X 0,Y 114.586,Z 404.02,A -85,B 0,C 180,E1 -26299.719,E2 -26299.719} C_VEL
LIN {X 0,Y 119.316,Z 412.487,A -85,B 0,C 180,E1 -26305.285,E2 -26305.285} C_VEL
LIN {X 0,Y 125.468,Z 419.442,A -85,B 0,C 180,E1 -26310.278,E2 -26310.278} C_VEL
LIN {X 0,Y 134.082,Z 425.666,A -85,B 0,C 180,E1 -26315.214,E2 -26315.214} C_VEL
LIN {X 0,Y 144.005,Z 430.199,A -85,B 0,C 180,E1 -26319.383,E2 -26319.383} C_VEL
LIN {X 0,Y 146.88,Z 431.151,A -85,B 0,C 180,E1 -26320.409,E2 -26320.409} C_VEL
LIN {X 0,Y 146.331,Z 431.381,A -85,B 0,C 180,E1 -26321.249,E2 -26321.249} C_VEL
LIN {X 0,Y 138.176,Z 430.698,A -85,B 0,C 180,E1 -26324.596,E2 -26324.596} C_VEL
LIN {X 0,Y 129.159,Z 429.021,A -85,B 0,C 180,E1 -26329.628,E2 -26329.628} C_VEL
LIN {X 0,Y 122.471,Z 426.661,A -85,B 0,C 180,E1 -26334.981,E2 -26334.981} C_VEL
LIN {X 0,Y 117.272,Z 423.367,A -85,B 0,C 180,E1 -26341.352,E2 -26341.352} C_VEL
LIN {X 0,Y 114.019,Z 418.449,A -85,B 0,C 180,E1 -26349.344,E2 -26349.344} C_VEL
LIN {X 0,Y 113.862,Z 412.227,A -85,B 0,C 180,E1 -26357.524,E2 -26357.524} C_VEL
LIN {X 0,Y 115.27,Z 406.947,A -85,B 0,C 180,E1 -26362.996,E2 -26362.996} C_VEL
LIN {X 0,Y 116.458,Z 402.508,A -85,B 0,C 180,E1 -26366.54,E2 -26366.54} C_VEL
LIN {X 0,Y 118.695,Z 395.495,A -85,B 0,C 180,E1 -26371.111,E2 -26371.111} C_VEL
LIN {X 0,Y 121.739,Z 390.573,A -85,B 0,C 180,E1 -26374.175,E2 -26374.175} C_VEL
LIN {X 0,Y 123.791,Z 388.525,A -85,B 0,C 180,E1 -26375.645,E2 -26375.645} C_VEL
LIN {X 0,Y 120.922,Z 395.028,A -85,B 0,C 180,E1 -26378.846,E2 -26378.846} C_VEL
LIN {X 0,Y 118.777,Z 401.602,A -85,B 0,C 180,E1 -26382.809,E2 -26382.809} C_VEL
LIN {X 0,Y 117.316,Z 408.8,A -85,B 0,C 180,E1 -26388.331,E2 -26388.331} C_VEL
LIN {X 0,Y 117.962,Z 415.486,A -85,B 0,C 180,E1 -26394.648,E2 -26394.648} C_VEL
LIN {X 0,Y 121.481,Z 421.436,A -85,B 0,C 180,E1 -26401.378,E2 -26401.378} C_VEL
LIN {X 0,Y 127.512,Z 425.932,A -85,B 0,C 180,E1 -26407.321,E2 -26407.321} C_VEL
LIN {X 0,Y 131.295,Z 427.677,A -85,B 0,C 180,E1 -26409.967,E2 -26409.967} C_VEL
LIN {X 0,Y 135.588,Z 429.104,A -85,B 0,C 180,E1 -26412.364,E2 -26412.364} C_VEL
LIN {X 0,Y 140.275,Z 430.161,A -85,B 0,C 180,E1 -26414.541,E2 -26414.541} C_VEL
LIN {X 0,Y 145.33,Z 430.889,A -85,B 0,C 180,E1 -26416.501,E2 -26416.501} C_VEL
LIN {X 0,Y 150.752,Z 431.314,A -85,B 0,C 180,E1 -26418.238,E2 -26418.238} C_VEL
LIN {X 0,Y 149.605,Z 430.926,A -85,B 0,C 180,E1 -26418.873,E2 -26418.873} C_VEL
LIN {X 0,Y 141.643,Z 427.956,A -85,B 0,C 180,E1 -26421.663,E2 -26421.663} C_VEL
LIN {X 0,Y 134.334,Z 423.842,A -85,B 0,C 180,E1 -26424.862,E2 -26424.862} C_VEL
LIN {X 0,Y 127.831,Z 418.455,A -85,B 0,C 180,E1 -26428.509,E2 -26428.509} C_VEL
LIN {X 0,Y 123.177,Z 412.924,A -85,B 0,C 180,E1 -26431.915,E2 -26431.915} C_VEL
LIN {X 0,Y 118.637,Z 404.861,A -85,B 0,C 180,E1 -26436.426,E2 -26436.426} C_VEL
LIN {X 0,Y 115.884,Z 396.702,A -85,B 0,C 180,E1 -26440.511,E2 -26440.511} C_VEL
LIN {X 0,Y 114.334,Z 386.804,A -85,B 0,C 180,E1 -26444.852,E2 -26444.852} C_VEL
LIN {X 0,Y 113.97,Z 376.986,A -85,B 0,C 180,E1 -26448.434,E2 -26448.434} C_VEL
LIN {X 0,Y 114.183,Z 366.512,A -85,B 0,C 180,E1 -26451.523,E2 -26451.523} C_VEL
LIN {X 0,Y 110.322,Z 358.359,A -85,B 0,C 180,E1 -26458.17,E2 -26458.17} C_VEL
LIN {X 0,Y 107.036,Z 346.797,A -85,B 0,C 180,E1 -26468.383,E2 -26468.383} C_VEL
LIN {X 0,Y 106.152,Z 344.756,A -85,B 0,C 180,E1 -26470.146,E2 -26470.146} C_VEL
LIN {X 0,Y 103.195,Z 341.374,A -85,B 0,C 180,E1 -26472.874,E2 -26472.874} C_VEL
LIN {X 0,Y 100.352,Z 337.948,A -85,B 0,C 180,E1 -26475.752,E2 -26475.752} C_VEL
LIN {X 0,Y 99.71,Z 335.883,A -85,B 0,C 180,E1 -26477.688,E2 -26477.688} C_VEL
LIN {X 0,Y 99.84,Z 332.052,A -85,B 0,C 180,E1 -26481.552,E2 -26481.552} C_VEL
LIN {X 0,Y 100.465,Z 331.971,A -85,B 0,C 180,E1 -26489.313,E2 -26489.313} C_VEL
LIN {X 0,Y 100.656,Z 331.938,A -85,B 0,C 180,E1 -26493.951,E2 -26493.951} C_VEL
LIN {X 0,Y 100.636,Z 331.948,A -85,B 0,C 180,E1 -26499.807,E2 -26499.807} C_VEL
LIN {X 0,Y 100.634,Z 331.949,A -85,B 0,C 180,E1 -26505.703,E2 -26505.703} C_VEL
LIN {X 0,Y 100.621,Z 331.944,A -85,B 0,C 180,E1 -26511.051,E2 -26511.051} C_VEL
LIN {X 0,Y 100.687,Z 331.942,A -85,B 0,C 180,E1 -26516.878,E2 -26516.878} C_VEL
LIN {X 0,Y 100.778,Z 331.931,A -85,B 0,C 180,E1 -26525.265,E2 -26525.265} C_VEL
LIN {X 0,Y 100.808,Z 331.922,A -85,B 0,C 180,E1 -26529.599,E2 -26529.599} C_VEL
LIN {X 0,Y 101.091,Z 331.885,A -85,B 0,C 180,E1 -26536.706,E2 -26536.706} C_VEL
LIN {X 0,Y 101.225,Z 331.877,A -85,B 0,C 180,E1 -26542.018,E2 -26542.018} C_VEL
LIN {X 0,Y 101.817,Z 331.803,A -85,B 0,C 180,E1 -26550,E2 -26550} C_VEL
LIN {X 0,Y 101.225,Z 331.877,A -85,B 0,C 180,E1 -26557.982,E2 -26557.982} C_VEL
LIN {X 0,Y 101.091,Z 331.885,A -85,B 0,C 180,E1 -26563.294,E2 -26563.294} C_VEL
LIN {X 0,Y 100.825,Z 331.92,A -85,B 0,C 180,E1 -26570.397,E2 -26570.397} C_VEL
LIN {X 0,Y 100.766,Z 331.933,A -85,B 0,C 180,E1 -26574.961,E2 -26574.961} C_VEL
LIN {X 0,Y 100.689,Z 331.942,A -85,B 0,C 180,E1 -26583.124,E2 -26583.124} C_VEL
LIN {X 0,Y 100.632,Z 331.945,A -85,B 0,C 180,E1 -26589.814,E2 -26589.814} C_VEL
LIN {X 0,Y 100.636,Z 331.945,A -85,B 0,C 180,E1 -26595.713,E2 -26595.713} C_VEL
LIN {X 0,Y 100.693,Z 331.943,A -85,B 0,C 180,E1 -26601.092,E2 -26601.092} C_VEL
LIN {X 0,Y 100.764,Z 331.927,A -85,B 0,C 180,E1 -26606.822,E2 -26606.822} C_VEL
LIN {X 0,Y 100.431,Z 331.976,A -85,B 0,C 180,E1 -26610.676,E2 -26610.676} C_VEL
LIN {X 0,Y 99.748,Z 332.163,A -85,B 0,C 180,E1 -26615.249,E2 -26615.249} C_VEL
LIN {X 0,Y 99.092,Z 335.913,A -85,B 0,C 180,E1 -26621.394,E2 -26621.394} C_VEL
LIN {X 0,Y 100.267,Z 343.735,A -85,B 0,C 180,E1 -26633.97,E2 -26633.97} C_VEL
LIN {X 0,Y 102.916,Z 346.997,A -85,B 0,C 180,E1 -26638.782,E2 -26638.782} C_VEL
LIN {X 0,Y 103.779,Z 352.915,A -85,B 0,C 180,E1 -26640.005,E2 -26640.005} C_VEL
LIN {X 0,Y 103.895,Z 364.654,A -85,B 0,C 180,E1 -26643.398,E2 -26643.398} C_VEL
LIN {X 0,Y 103.962,Z 374.984,A -85,B 0,C 180,E1 -26647.287,E2 -26647.287} C_VEL
LIN {X 0,Y 104.733,Z 386.37,A -85,B 0,C 180,E1 -26652.602,E2 -26652.602} C_VEL
LIN {X 0,Y 106.782,Z 396.678,A -85,B 0,C 180,E1 -26658.223,E2 -26658.223} C_VEL
LIN {X 0,Y 110.877,Z 406.519,A -85,B 0,C 180,E1 -26664.336,E2 -26664.336} C_VEL
LIN {X 0,Y 115.748,Z 413.605,A -85,B 0,C 180,E1 -26669.066,E2 -26669.066} C_VEL
LIN {X 0,Y 121.584,Z 419.53,A -85,B 0,C 180,E1 -26673.312,E2 -26673.312} C_VEL
LIN {X 0,Y 128.371,Z 424.506,A -85,B 0,C 180,E1 -26677.034,E2 -26677.034} C_VEL
LIN {X 0,Y 136.508,Z 428.76,A -85,B 0,C 180,E1 -26680.508,E2 -26680.508} C_VEL
LIN {X 0,Y 135.314,Z 428.89,A -85,B 0,C 180,E1 -26681.719,E2 -26681.719} C_VEL
LIN {X 0,Y 124.565,Z 426.581,A -85,B 0,C 180,E1 -26687.386,E2 -26687.386} C_VEL
LIN {X 0,Y 117.21,Z 423.772,A -85,B 0,C 180,E1 -26693.158,E2 -26693.158} C_VEL
LIN {X 0,Y 110.756,Z 419.112,A -85,B 0,C 180,E1 -26701.581,E2 -26701.581} C_VEL
LIN {X 0,Y 108.149,Z 414.245,A -85,B 0,C 180,E1 -26709.058,E2 -26709.058} C_VEL
LIN {X 0,Y 108.164,Z 408.069,A -85,B 0,C 180,E1 -26717.085,E2 -26717.085} C_VEL
LIN {X 0,Y 109.912,Z 401.628,A -85,B 0,C 180,E1 -26723.575,E2 -26723.575} C_VEL
LIN {X 0,Y 112.032,Z 393.705,A -85,B 0,C 180,E1 -26729.192,E2 -26729.192} C_VEL
LIN {X 0,Y 114.328,Z 388.81,A -85,B 0,C 180,E1 -26732.308,E2 -26732.308} C_VEL
LIN {X 0,Y 117.634,Z 384.449,A -85,B 0,C 180,E1 -26735.058,E2 -26735.058} C_VEL
LIN {X 0,Y 119.406,Z 383.02,A -85,B 0,C 180,E1 -26736.175,E2 -26736.175} C_VEL
LIN {X 0,Y 116.792,Z 387.968,A -85,B 0,C 180,E1 -26738.617,E2 -26738.617} C_VEL
LIN {X 0,Y 114.545,Z 394.478,A -85,B 0,C 180,E1 -26742.175,E2 -26742.175} C_VEL
LIN {X 0,Y 112.802,Z 400.585,A -85,B 0,C 180,E1 -26746.402,E2 -26746.402} C_VEL
LIN {X 0,Y 112.143,Z 407.374,A -85,B 0,C 180,E1 -26752.088,E2 -26752.088} C_VEL
LIN {X 0,Y 113.642,Z 413.515,A -85,B 0,C 180,E1 -26758.223,E2 -26758.223} C_VEL
LIN {X 0,Y 117.675,Z 419.137,A -85,B 0,C 180,E1 -26764.567,E2 -26764.567} C_VEL
LIN {X 0,Y 122.524,Z 422.778,A -85,B 0,C 180,E1 -26769.121,E2 -26769.121} C_VEL
LIN {X 0,Y 126.394,Z 424.788,A -85,B 0,C 180,E1 -26771.855,E2 -26771.855} C_VEL
LIN {X 0,Y 130.786,Z 426.542,A -85,B 0,C 180,E1 -26774.313,E2 -26774.313} C_VEL
LIN {X 0,Y 138.878,Z 428.616,A -85,B 0,C 180,E1 -26777.844,E2 -26777.844} C_VEL
LIN {X 0,Y 139.799,Z 428.691,A -85,B 0,C 180,E1 -26778.468,E2 -26778.468} C_VEL
LIN {X 0,Y 133.563,Z 425.444,A -85,B 0,C 180,E1 -26780.84,E2 -26780.84} C_VEL
LIN {X 0,Y 125.229,Z 419.312,A -85,B 0,C 180,E1 -26784.879,E2 -26784.879} C_VEL
LIN {X 0,Y 119.125,Z 412.619,A -85,B 0,C 180,E1 -26788.916,E2 -26788.916} C_VEL
LIN {X 0,Y 114.908,Z 405.856,A -85,B 0,C 180,E1 -26792.691,E2 -26792.691} C_VEL
LIN {X 0,Y 111.017,Z 395.997,A -85,B 0,C 180,E1 -26797.672,E2 -26797.672} C_VEL
LIN {X 0,Y 109.266,Z 387.068,A -85,B 0,C 180,E1 -26801.721,E2 -26801.721} C_VEL
LIN {X 0,Y 108.59,Z 377.079,A -85,B 0,C 180,E1 -26805.573,E2 -26805.573} C_VEL
LIN {X 0,Y 108.529,Z 367.168,A -85,B 0,C 180,E1 -26808.793,E2 -26808.793} C_VEL
LIN {X 0,Y 104.649,Z 359.621,A -85,B 0,C 180,E1 -26815.18,E2 -26815.18} C_VEL
LIN {X 0,Y 99.68,Z 337.211,A -85,B 0,C 180,E1 -26836.375,E2 -26836.375} C_VEL
LIN {X 0,Y 99.71,Z 335.883,A -85,B 0,C 180,E1 -26837.688,E2 -26837.688} C_VEL
LIN {X 0,Y 99.429,Z 334.259,A -85,B 0,C 180,E1 -26839.709,E2 -26839.709} C_VEL
LIN {X 0,Y 98.224,Z 332.893,A -85,B 0,C 180,E1 -26842.945,E2 -26842.945} C_VEL
LIN {X 0,Y 96.022,Z 332.524,A -85,B 0,C 180,E1 -26847.486,E2 -26847.486} C_VEL
LIN {X 0,Y 93.791,Z 332.809,A -85,B 0,C 180,E1 -26853.604,E2 -26853.604} C_VEL
LIN {X 0,Y 93.513,Z 332.83,A -85,B 0,C 180,E1 -26856.134,E2 -26856.134} C_VEL
LIN {X 0,Y 93.523,Z 332.828,A -85,B 0,C 180,E1 -26862.549,E2 -26862.549} C_VEL
LIN {X 0,Y 93.526,Z 332.834,A -85,B 0,C 180,E1 -26868.707,E2 -26868.707} C_VEL
LIN {X 0,Y 93.583,Z 332.828,A -85,B 0,C 180,E1 -26875.688,E2 -26875.688} C_VEL
LIN {X 0,Y 93.66,Z 332.818,A -85,B 0,C 180,E1 -26884.203,E2 -26884.203} C_VEL
LIN {X 0,Y 93.684,Z 332.808,A -85,B 0,C 180,E1 -26887.97,E2 -26887.97} C_VEL
LIN {X 0,Y 94.011,Z 332.767,A -85,B 0,C 180,E1 -26896.345,E2 -26896.345} C_VEL
LIN {X 0,Y 94.16,Z 332.756,A -85,B 0,C 180,E1 -26901.415,E2 -26901.415} C_VEL
LIN {X 0,Y 94.746,Z 332.684,A -85,B 0,C 180,E1 -26910,E2 -26910} C_VEL
LIN {X 0,Y 94.16,Z 332.756,A -85,B 0,C 180,E1 -26918.585,E2 -26918.585} C_VEL
LIN {X 0,Y 94.011,Z 332.767,A -85,B 0,C 180,E1 -26923.655,E2 -26923.655} C_VEL
LIN {X 0,Y 93.695,Z 332.807,A -85,B 0,C 180,E1 -26932.027,E2 -26932.027} C_VEL
LIN {X 0,Y 93.615,Z 332.824,A -85,B 0,C 180,E1 -26936.772,E2 -26936.772} C_VEL
LIN {X 0,Y 93.584,Z 332.827,A -85,B 0,C 180,E1 -26944.313,E2 -26944.313} C_VEL
LIN {X 0,Y 93.523,Z 332.835,A -85,B 0,C 180,E1 -26952.558,E2 -26952.558} C_VEL
LIN {X 0,Y 93.556,Z 332.826,A -85,B 0,C 180,E1 -26958.695,E2 -26958.695} C_VEL
LIN {X 0,Y 93.66,Z 332.81,A -85,B 0,C 180,E1 -26965.631,E2 -26965.631} C_VEL
LIN {X 0,Y 93.529,Z 332.832,A -85,B 0,C 180,E1 -26968.272,E2 -26968.272} C_VEL
LIN {X 0,Y 92.961,Z 332.904,A -85,B 0,C 180,E1 -26973.031,E2 -26973.031} C_VEL
LIN {X 0,Y 92.484,Z 333.019,A -85,B 0,C 180,E1 -26976.623,E2 -26976.623} C_VEL
LIN {X 0,Y 93.707,Z 344.015,A -85,B 0,C 180,E1 -26995.704,E2 -26995.704} C_VEL
LIN {X 0,Y 96.788,Z 347.361,A -85,B 0,C 180,E1 -27000.85,E2 -27000.85} C_VEL
LIN {X 0,Y 97.47,Z 352.08,A -85,B 0,C 180,E1 -27001.813,E2 -27001.813} C_VEL
LIN {X 0,Y 97.726,Z 363.015,A -85,B 0,C 180,E1 -27005.163,E2 -27005.163} C_VEL
LIN {X 0,Y 97.926,Z 373.455,A -85,B 0,C 180,E1 -27009.298,E2 -27009.298} C_VEL
LIN {X 0,Y 98.812,Z 384.223,A -85,B 0,C 180,E1 -27014.42,E2 -27014.42} C_VEL
LIN {X 0,Y 101.124,Z 394.742,A -85,B 0,C 180,E1 -27020.339,E2 -27020.339} C_VEL
LIN {X 0,Y 105.57,Z 405.045,A -85,B 0,C 180,E1 -27026.708,E2 -27026.708} C_VEL
LIN {X 0,Y 111.719,Z 413.474,A -85,B 0,C 180,E1 -27032.33,E2 -27032.33} C_VEL
LIN {X 0,Y 118.068,Z 419.538,A -85,B 0,C 180,E1 -27036.535,E2 -27036.535} C_VEL
LIN {X 0,Y 126.47,Z 425.296,A -85,B 0,C 180,E1 -27040.657,E2 -27040.657} C_VEL
LIN {X 0,Y 125.752,Z 425.484,A -85,B 0,C 180,E1 -27041.924,E2 -27041.924} C_VEL
LIN {X 0,Y 115.819,Z 422.342,A -85,B 0,C 180,E1 -27048.126,E2 -27048.126} C_VEL
LIN {X 0,Y 109.054,Z 418.758,A -85,B 0,C 180,E1 -27054.549,E2 -27054.549} C_VEL
LIN {X 0,Y 103.892,Z 413.45,A -85,B 0,C 180,E1 -27063.359,E2 -27063.359} C_VEL
LIN {X 0,Y 102.232,Z 407.381,A -85,B 0,C 180,E1 -27071.979,E2 -27071.979} C_VEL
LIN {X 0,Y 103.324,Z 400.708,A -85,B 0,C 180,E1 -27079.806,E2 -27079.806} C_VEL
LIN {X 0,Y 104.713,Z 395.809,A -85,B 0,C 180,E1 -27084.222,E2 -27084.222} C_VEL
LIN {X 0,Y 107.27,Z 387.406,A -85,B 0,C 180,E1 -27090,E2 -27090} C_VEL
LIN {X 0,Y 110.697,Z 381.759,A -85,B 0,C 180,E1 -27093.64,E2 -27093.64} C_VEL
LIN {X 0,Y 114.434,Z 377.871,A -85,B 0,C 180,E1 -27096.159,E2 -27096.159} C_VEL
LIN {X 0,Y 114.574,Z 377.794,A -85,B 0,C 180,E1 -27096.251,E2 -27096.251} C_VEL
LIN {X 0,Y 113.782,Z 379.585,A -85,B 0,C 180,E1 -27097.982,E2 -27097.982} C_VEL
LIN {X 0,Y 109.994,Z 389.105,A -85,B 0,C 180,E1 -27102.924,E2 -27102.924} C_VEL
LIN {X 0,Y 107.876,Z 396.546,A -85,B 0,C 180,E1 -27108.09,E2 -27108.09} C_VEL
LIN {X 0,Y 107.35,Z 402.961,A -85,B 0,C 180,E1 -27113.563,E2 -27113.563} C_VEL
LIN {X 0,Y 108.718,Z 409.205,A -85,B 0,C 180,E1 -27119.626,E2 -27119.626} C_VEL
LIN {X 0,Y 112.677,Z 415.143,A -85,B 0,C 180,E1 -27126.116,E2 -27126.116} C_VEL
LIN {X 0,Y 119.699,Z 420.545,A -85,B 0,C 180,E1 -27132.471,E2 -27132.471} C_VEL
LIN {X 0,Y 127.996,Z 424.252,A -85,B 0,C 180,E1 -27137.222,E2 -27137.222} C_VEL
LIN {X 0,Y 129.513,Z 424.672,A -85,B 0,C 180,E1 -27138.318,E2 -27138.318} C_VEL
LIN {X 0,Y 122.023,Z 419.002,A -85,B 0,C 180,E1 -27141.741,E2 -27141.741} C_VEL
LIN {X 0,Y 115.431,Z 412.098,A -85,B 0,C 180,E1 -27145.719,E2 -27145.719} C_VEL
LIN {X 0,Y 110.025,Z 403.651,A -85,B 0,C 180,E1 -27150.322,E2 -27150.322} C_VEL
LIN {X 0,Y 106.512,Z 395.077,A -85,B 0,C 180,E1 -27154.598,E2 -27154.598} C_VEL
LIN {X 0,Y 104.283,Z 384.859,A -85,B 0,C 180,E1 -27159.274,E2 -27159.274} C_VEL
LIN {X 0,Y 103.506,Z 376.172,A -85,B 0,C 180,E1 -27162.712,E2 -27162.712} C_VEL
LIN {X 0,Y 103.442,Z 368.124,A -85,B 0,C 180,E1 -27165.448,E2 -27165.448} C_VEL
LIN {X 0,Y 98.605,Z 359.677,A -85,B 0,C 180,E1 -27172.83,E2 -27172.83} C_VEL
LIN {X 0,Y 92.659,Z 336.024,A -85,B 0,C 180,E1 -27196.519,E2 -27196.519} C_VEL
LIN {X 0,Y 92.712,Z 332.937,A -85,B 0,C 180,E1 -27199.939,E2 -27199.939} C_VEL
LIN {X 0,Y 93.099,Z 332.886,A -85,B 0,C 180,E1 -27206.926,E2 -27206.926} C_VEL
LIN {X 0,Y 93.499,Z 332.836,A -85,B 0,C 180,E1 -27211.74,E2 -27211.74} C_VEL
LIN {X 0,Y 93.513,Z 332.83,A -85,B 0,C 180,E1 -27216.134,E2 -27216.134} C_VEL
LIN {X 0,Y 92.867,Z 332.927,A -85,B 0,C 180,E1 -27219.738,E2 -27219.738} C_VEL
LIN {X 0,Y 91.38,Z 333.126,A -85,B 0,C 180,E1 -27223.317,E2 -27223.317} C_VEL
LIN {X 0,Y 86.915,Z 333.671,A -85,B 0,C 180,E1 -27233.334,E2 -27233.334} C_VEL
LIN {X 0,Y 86.477,Z 333.707,A -85,B 0,C 180,E1 -27236.006,E2 -27236.006} C_VEL
LIN {X 0,Y 86.575,Z 333.701,A -85,B 0,C 180,E1 -27243.233,E2 -27243.233} C_VEL
LIN {X 0,Y 86.637,Z 333.692,A -85,B 0,C 180,E1 -27251.066,E2 -27251.066} C_VEL
LIN {X 0,Y 86.922,Z 333.651,A -85,B 0,C 180,E1 -27255.962,E2 -27255.962} C_VEL
LIN {X 0,Y 87.07,Z 333.639,A -85,B 0,C 180,E1 -27260.71,E2 -27260.71} C_VEL
LIN {X 0,Y 87.676,Z 333.565,A -85,B 0,C 180,E1 -27270,E2 -27270} C_VEL
LIN {X 0,Y 87.07,Z 333.639,A -85,B 0,C 180,E1 -27279.29,E2 -27279.29} C_VEL
LIN {X 0,Y 86.922,Z 333.651,A -85,B 0,C 180,E1 -27284.038,E2 -27284.038} C_VEL
LIN {X 0,Y 86.661,Z 333.689,A -85,B 0,C 180,E1 -27288.929,E2 -27288.929} C_VEL
LIN {X 0,Y 86.577,Z 333.7,A -85,B 0,C 180,E1 -27296.769,E2 -27296.769} C_VEL
LIN {X 0,Y 86.502,Z 333.708,A -85,B 0,C 180,E1 -27305.673,E2 -27305.673} C_VEL
LIN {X 0,Y 86.467,Z 333.715,A -85,B 0,C 180,E1 -27312.996,E2 -27312.996} C_VEL
LIN {X 0,Y 86.48,Z 333.71,A -85,B 0,C 180,E1 -27319.457,E2 -27319.457} C_VEL
LIN {X 0,Y 86.602,Z 333.689,A -85,B 0,C 180,E1 -27325.392,E2 -27325.392} C_VEL
LIN {X 0,Y 86.104,Z 333.761,A -85,B 0,C 180,E1 -27330.684,E2 -27330.684} C_VEL
LIN {X 0,Y 85.544,Z 333.828,A -85,B 0,C 180,E1 -27335.753,E2 -27335.753} C_VEL
LIN {X 0,Y 85.146,Z 334,A -85,B 0,C 180,E1 -27338.521,E2 -27338.521} C_VEL
LIN {X 0,Y 86.256,Z 342.952,A -85,B 0,C 180,E1 -27355.333,E2 -27355.333} C_VEL
LIN {X 0,Y 90.456,Z 347.424,A -85,B 0,C 180,E1 -27362.789,E2 -27362.789} C_VEL
LIN {X 0,Y 90.975,Z 348.052,A -85,B 0,C 180,E1 -27363.327,E2 -27363.327} C_VEL
LIN {X 0,Y 91.452,Z 352.574,A -85,B 0,C 180,E1 -27364.413,E2 -27364.413} C_VEL
LIN {X 0,Y 91.839,Z 364.078,A -85,B 0,C 180,E1 -27368.255,E2 -27368.255} C_VEL
LIN {X 0,Y 92.342,Z 375.418,A -85,B 0,C 180,E1 -27373.204,E2 -27373.204} C_VEL
LIN {X 0,Y 93.808,Z 385.572,A -85,B 0,C 180,E1 -27378.572,E2 -27378.572} C_VEL
LIN {X 0,Y 96.875,Z 395.971,A -85,B 0,C 180,E1 -27384.66,E2 -27384.66} C_VEL
LIN {X 0,Y 102.257,Z 405.96,A -85,B 0,C 180,E1 -27391.034,E2 -27391.034} C_VEL
LIN {X 0,Y 109.197,Z 414.352,A -85,B 0,C 180,E1 -27396.542,E2 -27396.542} C_VEL
LIN {X 0,Y 117.463,Z 421.247,A -85,B 0,C 180,E1 -27401.164,E2 -27401.164} C_VEL
LIN {X 0,Y 115.364,Z 420.803,A -85,B 0,C 180,E1 -27403.026,E2 -27403.026} C_VEL
LIN {X 0,Y 105.672,Z 416.275,A -85,B 0,C 180,E1 -27410.815,E2 -27410.815} C_VEL
LIN {X 0,Y 99.298,Z 410.509,A -85,B 0,C 180,E1 -27420.301,E2 -27420.301} C_VEL
LIN {X 0,Y 96.992,Z 404.755,A -85,B 0,C 180,E1 -27428.759,E2 -27428.759} C_VEL
LIN {X 0,Y 97.569,Z 397.692,A -85,B 0,C 180,E1 -27437.52,E2 -27437.52} C_VEL
LIN {X 0,Y 98.762,Z 393.437,A -85,B 0,C 180,E1 -27441.818,E2 -27441.818} C_VEL
LIN {X 0,Y 101.527,Z 383.673,A -85,B 0,C 180,E1 -27448.909,E2 -27448.909} C_VEL
LIN {X 0,Y 104.622,Z 378.15,A -85,B 0,C 180,E1 -27452.584,E2 -27452.584} C_VEL
LIN {X 0,Y 108.784,Z 373.364,A -85,B 0,C 180,E1 -27455.757,E2 -27455.757} C_VEL
LIN {X 0,Y 107.531,Z 376.7,A -85,B 0,C 180,E1 -27459.345,E2 -27459.345} C_VEL
LIN {X 0,Y 107.359,Z 378.816,A -85,B 0,C 180,E1 -27461.326,E2 -27461.326} C_VEL
LIN {X 0,Y 104.82,Z 386.281,A -85,B 0,C 180,E1 -27465.557,E2 -27465.557} C_VEL
LIN {X 0,Y 103.077,Z 393.47,A -85,B 0,C 180,E1 -27470.893,E2 -27470.893} C_VEL
LIN {X 0,Y 103.087,Z 401.004,A -85,B 0,C 180,E1 -27477.581,E2 -27477.581} C_VEL
LIN {X 0,Y 105.807,Z 407.918,A -85,B 0,C 180,E1 -27484.634,E2 -27484.634} C_VEL
LIN {X 0,Y 111.327,Z 414.004,A -85,B 0,C 180,E1 -27491.278,E2 -27491.278} C_VEL
LIN {X 0,Y 118.892,Z 418.921,A -85,B 0,C 180,E1 -27496.833,E2 -27496.833} C_VEL
LIN {X 0,Y 120.01,Z 419.268,A -85,B 0,C 180,E1 -27498.08,E2 -27498.08} C_VEL
LIN {X 0,Y 113.285,Z 412.651,A -85,B 0,C 180,E1 -27501.651,E2 -27501.651} C_VEL
LIN {X 0,Y 107.175,Z 404.32,A -85,B 0,C 180,E1 -27506.119,E2 -27506.119} C_VEL
LIN {X 0,Y 102.447,Z 394.018,A -85,B 0,C 180,E1 -27511.295,E2 -27511.295} C_VEL
LIN {X 0,Y 99.985,Z 384.647,A -85,B 0,C 180,E1 -27515.604,E2 -27515.604} C_VEL
LIN {X 0,Y 98.804,Z 374.115,A -85,B 0,C 180,E1 -27519.888,E2 -27519.888} C_VEL
LIN {X 0,Y 98.586,Z 368.858,A -85,B 0,C 180,E1 -27521.826,E2 -27521.826} C_VEL
LIN {X 0,Y 92.659,Z 359.403,A -85,B 0,C 180,E1 -27530.411,E2 -27530.411} C_VEL
LIN {X 0,Y 85.648,Z 335.802,A -85,B 0,C 180,E1 -27555.461,E2 -27555.461} C_VEL
LIN {X 0,Y 85.622,Z 333.823,A -85,B 0,C 180,E1 -27557.921,E2 -27557.921} C_VEL
LIN {X 0,Y 85.983,Z 333.77,A -85,B 0,C 180,E1 -27565.958,E2 -27565.958} C_VEL
LIN {X 0,Y 86.184,Z 333.75,A -85,B 0,C 180,E1 -27569.286,E2 -27569.286} C_VEL
LIN {X 0,Y 86.479,Z 333.705,A -85,B 0,C 180,E1 -27575.942,E2 -27575.942} C_VEL
LIN {X 0,Y 86.467,Z 333.706,A -85,B 0,C 180,E1 -27582.986,E2 -27582.986} C_VEL
LIN {X 0,Y 86.449,Z 333.713,A -85,B 0,C 180,E1 -27589.43,E2 -27589.43} C_VEL
LIN {X 0,Y 86.477,Z 333.707,A -85,B 0,C 180,E1 -27596.006,E2 -27596.006} C_VEL
LIN {X 0,Y 85.666,Z 333.808,A -85,B 0,C 180,E1 -27599.898,E2 -27599.898} C_VEL
LIN {X 0,Y 84.118,Z 334.007,A -85,B 0,C 180,E1 -27603.772,E2 -27603.772} C_VEL
LIN {X 0,Y 80.031,Z 334.513,A -85,B 0,C 180,E1 -27614.687,E2 -27614.687} C_VEL
LIN {X 0,Y 79.824,Z 334.531,A -85,B 0,C 180,E1 -27617.584,E2 -27617.584} C_VEL
LIN {X 0,Y 80.089,Z 334.501,A -85,B 0,C 180,E1 -27624.966,E2 -27624.966} C_VEL
LIN {X 0,Y 80.606,Z 334.445,A -85,B 0,C 180,E1 -27630,E2 -27630} C_VEL
LIN {X 0,Y 79.954,Z 334.524,A -85,B 0,C 180,E1 -27640.125,E2 -27640.125} C_VEL
LIN {X 0,Y 79.74,Z 334.55,A -85,B 0,C 180,E1 -27645.332,E2 -27645.332} C_VEL
LIN {X 0,Y 79.519,Z 334.572,A -85,B 0,C 180,E1 -27650.703,E2 -27650.703} C_VEL
LIN {X 0,Y 79.475,Z 334.582,A -85,B 0,C 180,E1 -27657.849,E2 -27657.849} C_VEL
LIN {X 0,Y 79.373,Z 334.595,A -85,B 0,C 180,E1 -27662.091,E2 -27662.091} C_VEL
LIN {X 0,Y 79.359,Z 334.591,A -85,B 0,C 180,E1 -27668.311,E2 -27668.311} C_VEL
LIN {X 0,Y 79.404,Z 334.59,A -85,B 0,C 180,E1 -27675.079,E2 -27675.079} C_VEL
LIN {X 0,Y 79.452,Z 334.587,A -85,B 0,C 180,E1 -27682.759,E2 -27682.759} C_VEL
LIN {X 0,Y 79.237,Z 334.612,A -85,B 0,C 180,E1 -27687.856,E2 -27687.856} C_VEL
LIN {X 0,Y 78.691,Z 334.68,A -85,B 0,C 180,E1 -27693.485,E2 -27693.485} C_VEL
LIN {X 0,Y 77.814,Z 335.006,A -85,B 0,C 180,E1 -27700.896,E2 -27700.896} C_VEL
LIN {X 0,Y 79.772,Z 343.125,A -85,B 0,C 180,E1 -27717.482,E2 -27717.482} C_VEL
LIN {X 0,Y 84.055,Z 347.291,A -85,B 0,C 180,E1 -27724.802,E2 -27724.802} C_VEL
LIN {X 0,Y 85.221,Z 348.122,A -85,B 0,C 180,E1 -27726.048,E2 -27726.048} C_VEL
LIN {X 0,Y 85.683,Z 353.955,A -85,B 0,C 180,E1 -27727.664,E2 -27727.664} C_VEL
LIN {X 0,Y 86.066,Z 362.127,A -85,B 0,C 180,E1 -27730.594,E2 -27730.594} C_VEL
LIN {X 0,Y 87.007,Z 374.665,A -85,B 0,C 180,E1 -27736.428,E2 -27736.428} C_VEL
LIN {X 0,Y 88.854,Z 385.008,A -85,B 0,C 180,E1 -27742.074,E2 -27742.074} C_VEL
LIN {X 0,Y 92.496,Z 395.292,A -85,B 0,C 180,E1 -27748.358,E2 -27748.358} C_VEL
LIN {X 0,Y 98.55,Z 405.538,A -85,B 0,C 180,E1 -27754.792,E2 -27754.792} C_VEL
LIN {X 0,Y 107.322,Z 415.062,A -85,B 0,C 180,E1 -27760.914,E2 -27760.914} C_VEL
LIN {X 0,Y 108.636,Z 416.196,A -85,B 0,C 180,E1 -27761.629,E2 -27761.629} C_VEL
LIN {X 0,Y 107.973,Z 416.197,A -85,B 0,C 180,E1 -27762.814,E2 -27762.814} C_VEL
LIN {X 0,Y 99.406,Z 411.411,A -85,B 0,C 180,E1 -27770.483,E2 -27770.483} C_VEL
LIN {X 0,Y 94.351,Z 406.384,A -85,B 0,C 180,E1 -27778.573,E2 -27778.573} C_VEL
LIN {X 0,Y 91.856,Z 400.3,A -85,B 0,C 180,E1 -27787.508,E2 -27787.508} C_VEL
LIN {X 0,Y 92.404,Z 392.93,A -85,B 0,C 180,E1 -27796.81,E2 -27796.81} C_VEL
LIN {X 0,Y 93.618,Z 388.356,A -85,B 0,C 180,E1 -27801.365,E2 -27801.365} C_VEL
LIN {X 0,Y 96.025,Z 379.597,A -85,B 0,C 180,E1 -27807.817,E2 -27807.817} C_VEL
LIN {X 0,Y 99.216,Z 373.743,A -85,B 0,C 180,E1 -27811.827,E2 -27811.827} C_VEL
LIN {X 0,Y 103.149,Z 368.949,A -85,B 0,C 180,E1 -27815.083,E2 -27815.083} C_VEL
LIN {X 0,Y 101.456,Z 373.506,A -85,B 0,C 180,E1 -27820.321,E2 -27820.321} C_VEL
LIN {X 0,Y 101.709,Z 377.933,A -85,B 0,C 180,E1 -27825.02,E2 -27825.02} C_VEL
LIN {X 0,Y 99.477,Z 385.328,A -85,B 0,C 180,E1 -27829.942,E2 -27829.942} C_VEL
LIN {X 0,Y 98.57,Z 393.212,A -85,B 0,C 180,E1 -27836.577,E2 -27836.577} C_VEL
LIN {X 0,Y 100.361,Z 400.945,A -85,B 0,C 180,E1 -27844.071,E2 -27844.071} C_VEL
LIN {X 0,Y 103.981,Z 406.571,A -85,B 0,C 180,E1 -27849.949,E2 -27849.949} C_VEL
LIN {X 0,Y 110.632,Z 412.474,A -85,B 0,C 180,E1 -27856.192,E2 -27856.192} C_VEL
LIN {X 0,Y 111.383,Z 412.682,A -85,B 0,C 180,E1 -27857.691,E2 -27857.691} C_VEL
LIN {X 0,Y 105.028,Z 404.722,A -85,B 0,C 180,E1 -27861.753,E2 -27861.753} C_VEL
LIN {X 0,Y 99.509,Z 394.591,A -85,B 0,C 180,E1 -27866.808,E2 -27866.808} C_VEL
LIN {X 0,Y 96.257,Z 384.209,A -85,B 0,C 180,E1 -27871.66,E2 -27871.66} C_VEL
LIN {X 0,Y 94.687,Z 374.266,A -85,B 0,C 180,E1 -27875.898,E2 -27875.898} C_VEL
LIN {X 0,Y 94.303,Z 369.655,A -85,B 0,C 180,E1 -27877.684,E2 -27877.684} C_VEL
LIN {X 0,Y 87.214,Z 359.496,A -85,B 0,C 180,E1 -27887.185,E2 -27887.185} C_VEL
LIN {X 0,Y 78.657,Z 334.793,A -85,B 0,C 180,E1 -27915.043,E2 -27915.043} C_VEL
LIN {X 0,Y 78.956,Z 334.645,A -85,B 0,C 180,E1 -27926.419,E2 -27926.419} C_VEL
LIN {X 0,Y 79.235,Z 334.612,A -85,B 0,C 180,E1 -27932.145,E2 -27932.145} C_VEL
LIN {X 0,Y 79.359,Z 334.6,A -85,B 0,C 180,E1 -27938.301,E2 -27938.301} C_VEL
LIN {X 0,Y 79.378,Z 334.594,A -85,B 0,C 180,E1 -27945.087,E2 -27945.087} C_VEL
LIN {X 0,Y 79.379,Z 334.591,A -85,B 0,C 180,E1 -27952.817,E2 -27952.817} C_VEL
LIN {X 0,Y 79.371,Z 334.595,A -85,B 0,C 180,E1 -27957.908,E2 -27957.908} C_VEL
LIN {X 0,Y 79.516,Z 334.58,A -85,B 0,C 180,E1 -27963.773,E2 -27963.773} C_VEL
LIN {X 0,Y 79.504,Z 334.574,A -85,B 0,C 180,E1 -27969.293,E2 -27969.293} C_VEL
LIN {X 0,Y 79.815,Z 334.538,A -85,B 0,C 180,E1 -27975.572,E2 -27975.572} C_VEL
LIN {X 0,Y 79.824,Z 334.531,A -85,B 0,C 180,E1 -27977.584,E2 -27977.584} C_VEL
LIN {X 0,Y 79.597,Z 334.57,A -85,B 0,C 180,E1 -27980.41,E2 -27980.41} C_VEL
LIN {X 0,Y 78.403,Z 334.721,A -85,B 0,C 180,E1 -27984.628,E2 -27984.628} C_VEL
LIN {X 0,Y 75.384,Z 335.107,A -85,B 0,C 180,E1 -27991.803,E2 -27991.803} C_VEL
LIN {X 0,Y 72.845,Z 335.406,A -85,B 0,C 180,E1 -28001.142,E2 -28001.142} C_VEL
LIN {X 0,Y 72.571,Z 335.445,A -85,B 0,C 180,E1 -28006.89,E2 -28006.89} C_VEL
LIN {X 0,Y 72.394,Z 335.461,A -85,B 0,C 180,E1 -28012.85,E2 -28012.85} C_VEL
LIN {X 0,Y 72.369,Z 335.463,A -85,B 0,C 180,E1 -28019.086,E2 -28019.086} C_VEL
LIN {X 0,Y 72.288,Z 335.479,A -85,B 0,C 180,E1 -28025.686,E2 -28025.686} C_VEL
LIN {X 0,Y 72.253,Z 335.486,A -85,B 0,C 180,E1 -28032.913,E2 -28032.913} C_VEL
LIN {X 0,Y 72.338,Z 335.475,A -85,B 0,C 180,E1 -28041.009,E2 -28041.009} C_VEL
LIN {X 0,Y 72.268,Z 335.476,A -85,B 0,C 180,E1 -28044.313,E2 -28044.313} C_VEL
LIN {X 0,Y 71.765,Z 335.544,A -85,B 0,C 180,E1 -28051.81,E2 -28051.81} C_VEL
LIN {X 0,Y 71.141,Z 335.623,A -85,B 0,C 180,E1 -28056.733,E2 -28056.733} C_VEL
LIN {X 0,Y 70.603,Z 335.784,A -85,B 0,C 180,E1 -28063.378,E2 -28063.378} C_VEL
LIN {X 0,Y 73.399,Z 343.311,A -85,B 0,C 180,E1 -28080.007,E2 -28080.007} C_VEL
LIN {X 0,Y 77.947,Z 347.227,A -85,B 0,C 180,E1 -28087.339,E2 -28087.339} C_VEL
LIN {X 0,Y 79.883,Z 348.701,A -85,B 0,C 180,E1 -28089.341,E2 -28089.341} C_VEL
LIN {X 0,Y 80.53,Z 358.466,A -85,B 0,C 180,E1 -28092.741,E2 -28092.741} C_VEL
LIN {X 0,Y 81.522,Z 370.498,A -85,B 0,C 180,E1 -28098.283,E2 -28098.283} C_VEL
LIN {X 0,Y 83.256,Z 380.224,A -85,B 0,C 180,E1 -28103.645,E2 -28103.645} C_VEL
LIN {X 0,Y 87.04,Z 391.256,A -85,B 0,C 180,E1 -28110.315,E2 -28110.315} C_VEL
LIN {X 0,Y 92.252,Z 400.662,A -85,B 0,C 180,E1 -28116.193,E2 -28116.193} C_VEL
LIN {X 0,Y 99.901,Z 409.972,A -85,B 0,C 180,E1 -28121.944,E2 -28121.944} C_VEL
LIN {X 0,Y 100.581,Z 410.845,A -85,B 0,C 180,E1 -28122.902,E2 -28122.902} C_VEL
LIN {X 0,Y 92.996,Z 405.747,A -85,B 0,C 180,E1 -28130.853,E2 -28130.853} C_VEL
LIN {X 0,Y 88.662,Z 400.521,A -85,B 0,C 180,E1 -28138.987,E2 -28138.987} C_VEL
LIN {X 0,Y 86.783,Z 393.031,A -85,B 0,C 180,E1 -28149.718,E2 -28149.718} C_VEL
LIN {X 0,Y 87.776,Z 386.711,A -85,B 0,C 180,E1 -28157.325,E2 -28157.325} C_VEL
LIN {X 0,Y 88.663,Z 382.95,A -85,B 0,C 180,E1 -28160.878,E2 -28160.878} C_VEL
LIN {X 0,Y 91.44,Z 373.656,A -85,B 0,C 180,E1 -28167.795,E2 -28167.795} C_VEL
LIN {X 0,Y 94.977,Z 367.79,A -85,B 0,C 180,E1 -28171.908,E2 -28171.908} C_VEL
LIN {X 0,Y 97.683,Z 364.501,A -85,B 0,C 180,E1 -28174.126,E2 -28174.126} C_VEL
LIN {X 0,Y 95.906,Z 367.882,A -85,B 0,C 180,E1 -28178.428,E2 -28178.428} C_VEL
LIN {X 0,Y 95.46,Z 372.289,A -85,B 0,C 180,E1 -28183.722,E2 -28183.722} C_VEL
LIN {X 0,Y 96.411,Z 377.07,A -85,B 0,C 180,E1 -28189.455,E2 -28189.455} C_VEL
LIN {X 0,Y 94.765,Z 385.91,A -85,B 0,C 180,E1 -28196.422,E2 -28196.422} C_VEL
LIN {X 0,Y 95.636,Z 393.715,A -85,B 0,C 180,E1 -28203.675,E2 -28203.675} C_VEL
LIN {X 0,Y 99.603,Z 401.209,A -85,B 0,C 180,E1 -28211.31,E2 -28211.31} C_VEL
LIN {X 0,Y 103.611,Z 405.486,A -85,B 0,C 180,E1 -28215.684,E2 -28215.684} C_VEL
LIN {X 0,Y 104.242,Z 405.914,A -85,B 0,C 180,E1 -28216.817,E2 -28216.817} C_VEL
LIN {X 0,Y 98.225,Z 396.548,A -85,B 0,C 180,E1 -28221.365,E2 -28221.365} C_VEL
LIN {X 0,Y 93.727,Z 385.77,A -85,B 0,C 180,E1 -28226.42,E2 -28226.42} C_VEL
LIN {X 0,Y 91.324,Z 374.876,A -85,B 0,C 180,E1 -28231.243,E2 -28231.243} C_VEL
LIN {X 0,Y 90.674,Z 370.444,A -85,B 0,C 180,E1 -28233.079,E2 -28233.079} C_VEL
LIN {X 0,Y 81.876,Z 359.197,A -85,B 0,C 180,E1 -28243.795,E2 -28243.795} C_VEL
LIN {X 0,Y 71.756,Z 335.546,A -85,B 0,C 180,E1 -28272.134,E2 -28272.134} C_VEL
LIN {X 0,Y 71.605,Z 335.565,A -85,B 0,C 180,E1 -28283.108,E2 -28283.108} C_VEL
LIN {X 0,Y 71.984,Z 335.519,A -85,B 0,C 180,E1 -28289.211,E2 -28289.211} C_VEL
LIN {X 0,Y 72.225,Z 335.482,A -85,B 0,C 180,E1 -28295.712,E2 -28295.712} C_VEL
LIN {X 0,Y 72.239,Z 335.478,A -85,B 0,C 180,E1 -28302.913,E2 -28302.913} C_VEL
LIN {X 0,Y 72.286,Z 335.472,A -85,B 0,C 180,E1 -28311.047,E2 -28311.047} C_VEL
LIN {X 0,Y 72.287,Z 335.479,A -85,B 0,C 180,E1 -28314.314,E2 -28314.314} C_VEL
LIN {X 0,Y 72.367,Z 335.463,A -85,B 0,C 180,E1 -28320.949,E2 -28320.949} C_VEL
LIN {X 0,Y 72.385,Z 335.463,A -85,B 0,C 180,E1 -28327.147,E2 -28327.147} C_VEL
LIN {X 0,Y 72.712,Z 335.424,A -85,B 0,C 180,E1 -28335.108,E2 -28335.108} C_VEL
LIN {X 0,Y 72.846,Z 335.406,A -85,B 0,C 180,E1 -28338.875,E2 -28338.875} C_VEL
LIN {X 0,Y 73.535,Z 335.326,A -85,B 0,C 180,E1 -28350,E2 -28350} C_VEL
LIN {X 0,Y 72.845,Z 335.406,A -85,B 0,C 180,E1 -28361.142,E2 -28361.142} C_VEL
LIN {X 0,Y 72.327,Z 335.469,A -85,B 0,C 180,E1 -28364.216,E2 -28364.216} C_VEL
LIN {X 0,Y 70.749,Z 335.673,A -85,B 0,C 180,E1 -28368.788,E2 -28368.788} C_VEL
LIN {X 0,Y 67.336,Z 336.097,A -85,B 0,C 180,E1 -28376.64,E2 -28376.64} C_VEL
LIN {X 0,Y 65.332,Z 336.347,A -85,B 0,C 180,E1 -28383.484,E2 -28383.484} C_VEL
LIN {X 0,Y 65.053,Z 336.36,A -85,B 0,C 180,E1 -28387.059,E2 -28387.059} C_VEL
LIN {X 0,Y 65.183,Z 336.363,A -85,B 0,C 180,E1 -28391.011,E2 -28391.011} C_VEL
LIN {X 0,Y 65.237,Z 336.356,A -85,B 0,C 180,E1 -28399.742,E2 -28399.742} C_VEL
LIN {X 0,Y 64.908,Z 336.393,A -85,B 0,C 180,E1 -28407.232,E2 -28407.232} C_VEL
LIN {X 0,Y 64.797,Z 336.415,A -85,B 0,C 180,E1 -28410.193,E2 -28410.193} C_VEL
LIN {X 0,Y 64.344,Z 336.464,A -85,B 0,C 180,E1 -28414.103,E2 -28414.103} C_VEL
LIN {X 0,Y 63.521,Z 336.68,A -85,B 0,C 180,E1 -28426.818,E2 -28426.818} C_VEL
LIN {X 0,Y 67.231,Z 343.394,A -85,B 0,C 180,E1 -28443.004,E2 -28443.004} C_VEL
LIN {X 0,Y 74.732,Z 348.825,A -85,B 0,C 180,E1 -28453.175,E2 -28453.175} C_VEL
LIN {X 0,Y 75.501,Z 358.634,A -85,B 0,C 180,E1 -28456.919,E2 -28456.919} C_VEL
LIN {X 0,Y 76.789,Z 369.288,A -85,B 0,C 180,E1 -28462.189,E2 -28462.189} C_VEL
LIN {X 0,Y 79.658,Z 381.151,A -85,B 0,C 180,E1 -28469.036,E2 -28469.036} C_VEL
LIN {X 0,Y 83.416,Z 390.346,A -85,B 0,C 180,E1 -28474.667,E2 -28474.667} C_VEL
LIN {X 0,Y 90.43,Z 401.263,A -85,B 0,C 180,E1 -28481.353,E2 -28481.353} C_VEL
LIN {X 0,Y 92.706,Z 404.078,A -85,B 0,C 180,E1 -28483.029,E2 -28483.029} C_VEL
LIN {X 0,Y 90.889,Z 403.053,A -85,B 0,C 180,E1 -28485.899,E2 -28485.899} C_VEL
LIN {X 0,Y 84.385,Z 396.338,A -85,B 0,C 180,E1 -28496.403,E2 -28496.403} C_VEL
LIN {X 0,Y 82.082,Z 388.662,A -85,B 0,C 180,E1 -28507.559,E2 -28507.559} C_VEL
LIN {X 0,Y 83.086,Z 381.348,A -85,B 0,C 180,E1 -28516.597,E2 -28516.597} C_VEL
LIN {X 0,Y 84.251,Z 375.463,A -85,B 0,C 180,E1 -28521.727,E2 -28521.727} C_VEL
LIN {X 0,Y 87.136,Z 367.552,A -85,B 0,C 180,E1 -28527.686,E2 -28527.686} C_VEL
LIN {X 0,Y 92.272,Z 360.079,A -85,B 0,C 180,E1 -28533.087,E2 -28533.087} C_VEL
LIN {X 0,Y 90.429,Z 362.649,A -85,B 0,C 180,E1 -28536.695,E2 -28536.695} C_VEL
LIN {X 0,Y 89.431,Z 366.119,A -85,B 0,C 180,E1 -28541.33,E2 -28541.33} C_VEL
LIN {X 0,Y 90.908,Z 374.199,A -85,B 0,C 180,E1 -28551.905,E2 -28551.905} C_VEL
LIN {X 0,Y 91.771,Z 376.266,A -85,B 0,C 180,E1 -28554.713,E2 -28554.713} C_VEL
LIN {X 0,Y 91.472,Z 385.116,A -85,B 0,C 180,E1 -28562.536,E2 -28562.536} C_VEL
LIN {X 0,Y 93.8,Z 392.466,A -85,B 0,C 180,E1 -28569.704,E2 -28569.704} C_VEL
LIN {X 0,Y 95.568,Z 395.386,A -85,B 0,C 180,E1 -28572.652,E2 -28572.652} C_VEL
LIN {X 0,Y 97.297,Z 397.323,A -85,B 0,C 180,E1 -28576.247,E2 -28576.247} C_VEL
LIN {X 0,Y 92.555,Z 388.092,A -85,B 0,C 180,E1 -28580.503,E2 -28580.503} C_VEL
LIN {X 0,Y 89.05,Z 377.171,A -85,B 0,C 180,E1 -28585.434,E2 -28585.434} C_VEL
LIN {X 0,Y 87.74,Z 371.154,A -85,B 0,C 180,E1 -28588.093,E2 -28588.093} C_VEL
LIN {X 0,Y 76.016,Z 357.67,A -85,B 0,C 180,E1 -28601.113,E2 -28601.113} C_VEL
LIN {X 0,Y 65.049,Z 336.38,A -85,B 0,C 180,E1 -28628.358,E2 -28628.358} C_VEL
LIN {X 0,Y 64.412,Z 336.461,A -85,B 0,C 180,E1 -28639.098,E2 -28639.098} C_VEL
LIN {X 0,Y 64.936,Z 336.396,A -85,B 0,C 180,E1 -28650.021,E2 -28650.021} C_VEL
LIN {X 0,Y 65.175,Z 336.362,A -85,B 0,C 180,E1 -28660.989,E2 -28660.989} C_VEL
LIN {X 0,Y 65.194,Z 336.359,A -85,B 0,C 180,E1 -28669.698,E2 -28669.698} C_VEL
LIN {X 0,Y 65.246,Z 336.349,A -85,B 0,C 180,E1 -28679.494,E2 -28679.494} C_VEL
LIN {X 0,Y 65.231,Z 336.36,A -85,B 0,C 180,E1 -28684.471,E2 -28684.471} C_VEL
LIN {X 0,Y 65.616,Z 336.309,A -85,B 0,C 180,E1 -28694.541,E2 -28694.541} C_VEL
LIN {X 0,Y 65.744,Z 336.286,A -85,B 0,C 180,E1 -28697.655,E2 -28697.655} C_VEL
LIN {X 0,Y 66.435,Z 336.21,A -85,B 0,C 180,E1 -28710,E2 -28710} C_VEL
LIN {X 0,Y 65.753,Z 336.285,A -85,B 0,C 180,E1 -28722.343,E2 -28722.343} C_VEL
LIN {X 0,Y 65.378,Z 336.339,A -85,B 0,C 180,E1 -28728.814,E2 -28728.814} C_VEL
LIN {X 0,Y 65.235,Z 336.36,A -85,B 0,C 180,E1 -28735.527,E2 -28735.527} C_VEL
LIN {X 0,Y 65.188,Z 336.363,A -85,B 0,C 180,E1 -28742.62,E2 -28742.62} C_VEL
LIN {X 0,Y 65.053,Z 336.36,A -85,B 0,C 180,E1 -28747.059,E2 -28747.059} C_VEL
LIN {X 0,Y 64.751,Z 336.415,A -85,B 0,C 180,E1 -28750.512,E2 -28750.512} C_VEL
LIN {X 0,Y 63.355,Z 336.595,A -85,B 0,C 180,E1 -28755.658,E2 -28755.658} C_VEL
LIN {X 0,Y 61.36,Z 336.842,A -85,B 0,C 180,E1 -28760.836,E2 -28760.836} C_VEL
LIN {X 0,Y 56.892,Z 337.387,A -85,B 0,C 180,E1 -28776.392,E2 -28776.392} C_VEL
LIN {X 0,Y 56.766,Z 337.538,A -85,B 0,C 180,E1 -28791.194,E2 -28791.194} C_VEL
LIN {X 0,Y 61.288,Z 343.484,A -85,B 0,C 180,E1 -28806.593,E2 -28806.593} C_VEL
LIN {X 0,Y 70.027,Z 349.396,A -85,B 0,C 180,E1 -28817.78,E2 -28817.78} C_VEL
LIN {X 0,Y 70.94,Z 357.702,A -85,B 0,C 180,E1 -28821.299,E2 -28821.299} C_VEL
LIN {X 0,Y 73.08,Z 370.22,A -85,B 0,C 180,E1 -28827.891,E2 -28827.891} C_VEL
LIN {X 0,Y 76.009,Z 379.963,A -85,B 0,C 180,E1 -28833.703,E2 -28833.703} C_VEL
LIN {X 0,Y 81.406,Z 390.841,A -85,B 0,C 180,E1 -28840.361,E2 -28840.361} C_VEL
LIN {X 0,Y 85.722,Z 397.253,A -85,B 0,C 180,E1 -28844.116,E2 -28844.116} C_VEL
LIN {X 0,Y 83.692,Z 395.642,A -85,B 0,C 180,E1 -28847.794,E2 -28847.794} C_VEL
LIN {X 0,Y 78.977,Z 389.21,A -85,B 0,C 180,E1 -28857.729,E2 -28857.729} C_VEL
LIN {X 0,Y 77.71,Z 381.533,A -85,B 0,C 180,E1 -28868.792,E2 -28868.792} C_VEL
LIN {X 0,Y 78.696,Z 375.212,A -85,B 0,C 180,E1 -28876.247,E2 -28876.247} C_VEL
LIN {X 0,Y 81.509,Z 364.445,A -85,B 0,C 180,E1 -28885.054,E2 -28885.054} C_VEL
LIN {X 0,Y 85.283,Z 357.897,A -85,B 0,C 180,E1 -28890,E2 -28890} C_VEL
LIN {X 0,Y 87.017,Z 355.603,A -85,B 0,C 180,E1 -28891.736,E2 -28891.736} C_VEL
LIN {X 0,Y 84.336,Z 359.033,A -85,B 0,C 180,E1 -28896.94,E2 -28896.94} C_VEL
LIN {X 0,Y 83.39,Z 362.632,A -85,B 0,C 180,E1 -28902.163,E2 -28902.163} C_VEL
LIN {X 0,Y 85.498,Z 371.13,A -85,B 0,C 180,E1 -28914.268,E2 -28914.268} C_VEL
LIN {X 0,Y 88.197,Z 375.535,A -85,B 0,C 180,E1 -28920.865,E2 -28920.865} C_VEL
LIN {X 0,Y 89.516,Z 384.06,A -85,B 0,C 180,E1 -28928.909,E2 -28928.909} C_VEL
LIN {X 0,Y 92.354,Z 389.761,A -85,B 0,C 180,E1 -28934.742,E2 -28934.742} C_VEL
LIN {X 0,Y 88.029,Z 379.728,A -85,B 0,C 180,E1 -28939.174,E2 -28939.174} C_VEL
LIN {X 0,Y 85.836,Z 372.027,A -85,B 0,C 180,E1 -28942.548,E2 -28942.548} C_VEL
LIN {X 0,Y 71.293,Z 357.113,A -85,B 0,C 180,E1 -28956.769,E2 -28956.769} C_VEL
LIN {X 0,Y 58.717,Z 337.172,A -85,B 0,C 180,E1 -28983.422,E2 -28983.422} C_VEL
LIN {X 0,Y 57.452,Z 337.325,A -85,B 0,C 180,E1 -28994.152,E2 -28994.152} C_VEL
LIN {X 0,Y 57.359,Z 337.342,A -85,B 0,C 180,E1 -29001.556,E2 -29001.556} C_VEL
LIN {X 0,Y 57.803,Z 337.285,A -85,B 0,C 180,E1 -29009.09,E2 -29009.09} C_VEL
LIN {X 0,Y 57.934,Z 337.267,A -85,B 0,C 180,E1 -29017.329,E2 -29017.329} C_VEL
LIN {X 0,Y 58.004,Z 337.26,A -85,B 0,C 180,E1 -29026.621,E2 -29026.621} C_VEL
LIN {X 0,Y 58.023,Z 337.25,A -85,B 0,C 180,E1 -29032.726,E2 -29032.726} C_VEL
LIN {X 0,Y 58.15,Z 337.237,A -85,B 0,C 180,E1 -29037.764,E2 -29037.764} C_VEL
LIN {X 0,Y 58.142,Z 337.234,A -85,B 0,C 180,E1 -29041.085,E2 -29041.085} C_VEL
LIN {X 0,Y 58.508,Z 337.196,A -85,B 0,C 180,E1 -29053.905,E2 -29053.905} C_VEL
LIN {X 0,Y 58.777,Z 337.161,A -85,B 0,C 180,E1 -29063.133,E2 -29063.133} C_VEL
LIN {X 0,Y 59.33,Z 337.095,A -85,B 0,C 180,E1 -29070,E2 -29070} C_VEL
LIN {X 0,Y 58.779,Z 337.16,A -85,B 0,C 180,E1 -29076.867,E2 -29076.867} C_VEL
LIN {X 0,Y 58.521,Z 337.195,A -85,B 0,C 180,E1 -29086.141,E2 -29086.141} C_VEL
LIN {X 0,Y 58.144,Z 337.234,A -85,B 0,C 180,E1 -29098.914,E2 -29098.914} C_VEL
LIN {X 0,Y 58.025,Z 337.249,A -85,B 0,C 180,E1 -29107.17,E2 -29107.17} C_VEL
LIN {X 0,Y 58.032,Z 337.247,A -85,B 0,C 180,E1 -29116.605,E2 -29116.605} C_VEL
LIN {X 0,Y 57.937,Z 337.267,A -85,B 0,C 180,E1 -29122.673,E2 -29122.673} C_VEL
LIN {X 0,Y 57.812,Z 337.281,A -85,B 0,C 180,E1 -29128.317,E2 -29128.317} C_VEL
LIN {X 0,Y 57.612,Z 337.309,A -85,B 0,C 180,E1 -29130.805,E2 -29130.805} C_VEL
LIN {X 0,Y 56.892,Z 337.387,A -85,B 0,C 180,E1 -29136.392,E2 -29136.392} C_VEL
LIN {X 0,Y 55.953,Z 337.551,A -85,B 0,C 180,E1 -29140.353,E2 -29140.353} C_VEL
LIN {X 0,Y 53.006,Z 337.884,A -85,B 0,C 180,E1 -29146.828,E2 -29146.828} C_VEL
LIN {X 0,Y 50.691,Z 338.204,A -85,B 0,C 180,E1 -29153.855,E2 -29153.855} C_VEL
LIN {X 0,Y 50.691,Z 338.766,A -85,B 0,C 180,E1 -29157.872,E2 -29157.872} C_VEL
LIN {X 0,Y 50.76,Z 338.869,A -85,B 0,C 180,E1 -29158.214,E2 -29158.214} C_VEL
LIN {X 0,Y 55.671,Z 343.478,A -85,B 0,C 180,E1 -29170.925,E2 -29170.925} C_VEL
LIN {X 0,Y 65.863,Z 349.544,A -85,B 0,C 180,E1 -29182.972,E2 -29182.972} C_VEL
LIN {X 0,Y 67.223,Z 358.635,A -85,B 0,C 180,E1 -29187.286,E2 -29187.286} C_VEL
LIN {X 0,Y 69.621,Z 369.194,A -85,B 0,C 180,E1 -29193.127,E2 -29193.127} C_VEL
LIN {X 0,Y 73.963,Z 380.444,A -85,B 0,C 180,E1 -29199.904,E2 -29199.904} C_VEL
LIN {X 0,Y 79.101,Z 389.56,A -85,B 0,C 180,E1 -29205.308,E2 -29205.308} C_VEL
LIN {X 0,Y 78.316,Z 388.93,A -85,B 0,C 180,E1 -29208.029,E2 -29208.029} C_VEL
LIN {X 0,Y 73.996,Z 381.181,A -85,B 0,C 180,E1 -29219.931,E2 -29219.931} C_VEL
LIN {X 0,Y 73.676,Z 374.248,A -85,B 0,C 180,E1 -29229.682,E2 -29229.682} C_VEL
LIN {X 0,Y 74.376,Z 369.635,A -85,B 0,C 180,E1 -29234.901,E2 -29234.901} C_VEL
LIN {X 0,Y 76.811,Z 359.775,A -85,B 0,C 180,E1 -29243.206,E2 -29243.206} C_VEL
LIN {X 0,Y 80.239,Z 353.475,A -85,B 0,C 180,E1 -29248.227,E2 -29248.227} C_VEL
LIN {X 0,Y 80.456,Z 352.243,A -85,B 0,C 180,E1 -29252.065,E2 -29252.065} C_VEL
LIN {X 0,Y 78.067,Z 355.921,A -85,B 0,C 180,E1 -29257.954,E2 -29257.954} C_VEL
LIN {X 0,Y 77.349,Z 359.165,A -85,B 0,C 180,E1 -29263.13,E2 -29263.13} C_VEL
LIN {X 0,Y 79.957,Z 367.572,A -85,B 0,C 180,E1 -29276.071,E2 -29276.071} C_VEL
LIN {X 0,Y 85.906,Z 374.554,A -85,B 0,C 180,E1 -29287.481,E2 -29287.481} C_VEL
LIN {X 0,Y 87.022,Z 378.873,A -85,B 0,C 180,E1 -29291.582,E2 -29291.582} C_VEL
LIN {X 0,Y 87.488,Z 380.005,A -85,B 0,C 180,E1 -29293.691,E2 -29293.691} C_VEL
LIN {X 0,Y 85.019,Z 372.947,A -85,B 0,C 180,E1 -29296.731,E2 -29296.731} C_VEL
LIN {X 0,Y 67.071,Z 356.409,A -85,B 0,C 180,E1 -29311.858,E2 -29311.858} C_VEL
LIN {X 0,Y 55.091,Z 341.856,A -85,B 0,C 180,E1 -29330.815,E2 -29330.815} C_VEL
LIN {X 0,Y 52.871,Z 337.899,A -85,B 0,C 180,E1 -29337.609,E2 -29337.609} C_VEL
LIN {X 0,Y 50.286,Z 338.216,A -85,B 0,C 180,E1 -29356.221,E2 -29356.221} C_VEL
LIN {X 0,Y 50.373,Z 338.203,A -85,B 0,C 180,E1 -29364.732,E2 -29364.732} C_VEL
LIN {X 0,Y 50.817,Z 338.145,A -85,B 0,C 180,E1 -29373.922,E2 -29373.922} C_VEL
LIN {X 0,Y 50.971,Z 338.127,A -85,B 0,C 180,E1 -29383.569,E2 -29383.569} C_VEL
LIN {X 0,Y 51.021,Z 338.13,A -85,B 0,C 180,E1 -29395.72,E2 -29395.72} C_VEL
LIN {X 0,Y 51.014,Z 338.128,A -85,B 0,C 180,E1 -29405.588,E2 -29405.588} C_VEL
LIN {X 0,Y 51.449,Z 338.074,A -85,B 0,C 180,E1 -29414.145,E2 -29414.145} C_VEL
LIN {X 0,Y 51.657,Z 338.05,A -85,B 0,C 180,E1 -29422.181,E2 -29422.181} C_VEL
LIN {X 0,Y 52.218,Z 337.981,A -85,B 0,C 180,E1 -29430,E2 -29430} C_VEL
LIN {X 0,Y 51.661,Z 338.049,A -85,B 0,C 180,E1 -29437.819,E2 -29437.819} C_VEL
LIN {X 0,Y 51.388,Z 338.084,A -85,B 0,C 180,E1 -29446.834,E2 -29446.834} C_VEL
LIN {X 0,Y 51.017,Z 338.128,A -85,B 0,C 180,E1 -29454.411,E2 -29454.411} C_VEL
LIN {X 0,Y 51.022,Z 338.13,A -85,B 0,C 180,E1 -29464.282,E2 -29464.282} C_VEL
LIN {X 0,Y 51.007,Z 338.131,A -85,B 0,C 180,E1 -29473.545,E2 -29473.545} C_VEL
LIN {X 0,Y 51.001,Z 338.123,A -85,B 0,C 180,E1 -29476.463,E2 -29476.463} C_VEL
LIN {X 0,Y 50.748,Z 338.154,A -85,B 0,C 180,E1 -29486.374,E2 -29486.374} C_VEL
LIN {X 0,Y 49.908,Z 338.258,A -85,B 0,C 180,E1 -29495.385,E2 -29495.385} C_VEL
LIN {X 0,Y 50.391,Z 338.32,A -85,B 0,C 180,E1 -29516.512,E2 -29516.512} C_VEL
LIN {X 0,Y 50.76,Z 338.869,A -85,B 0,C 180,E1 -29518.214,E2 -29518.214} C_VEL
LIN {X 0,Y 51.197,Z 340.152,A -85,B 0,C 180,E1 -29522.475,E2 -29522.475} C_VEL
LIN {X 0,Y 51.754,Z 343.998,A -85,B 0,C 180,E1 -29536.93,E2 -29536.93} C_VEL
LIN {X 0,Y 53.639,Z 345.301,A -85,B 0,C 180,E1 -29540.422,E2 -29540.422} C_VEL
LIN {X 0,Y 60.824,Z 349.048,A -85,B 0,C 180,E1 -29547.537,E2 -29547.537} C_VEL
LIN {X 0,Y 62.48,Z 349.901,A -85,B 0,C 180,E1 -29549.027,E2 -29549.027} C_VEL
LIN {X 0,Y 64.976,Z 361.53,A -85,B 0,C 180,E1 -29555.099,E2 -29555.099} C_VEL
LIN {X 0,Y 69.021,Z 373.212,A -85,B 0,C 180,E1 -29561.939,E2 -29561.939} C_VEL
LIN {X 0,Y 72.848,Z 380.848,A -85,B 0,C 180,E1 -29566.363,E2 -29566.363} C_VEL
LIN {X 0,Y 73.563,Z 382.12,A -85,B 0,C 180,E1 -29568.029,E2 -29568.029} C_VEL
LIN {X 0,Y 69.752,Z 373.201,A -85,B 0,C 180,E1 -29581.648,E2 -29581.648} C_VEL
LIN {X 0,Y 70.05,Z 366.202,A -85,B 0,C 180,E1 -29590.97,E2 -29590.97} C_VEL
LIN {X 0,Y 71.938,Z 356.273,A -85,B 0,C 180,E1 -29600.013,E2 -29600.013} C_VEL
LIN {X 0,Y 73.177,Z 352.934,A -85,B 0,C 180,E1 -29602.966,E2 -29602.966} C_VEL
LIN {X 0,Y 72.898,Z 352.401,A -85,B 0,C 180,E1 -29604.468,E2 -29604.468} C_VEL
LIN {X 0,Y 73.475,Z 350.789,A -85,B 0,C 180,E1 -29610,E2 -29610} C_VEL
LIN {X 0,Y 73.527,Z 349.631,A -85,B 0,C 180,E1 -29613.552,E2 -29613.552} C_VEL
LIN {X 0,Y 71.486,Z 354.073,A -85,B 0,C 180,E1 -29621.34,E2 -29621.34} C_VEL
LIN {X 0,Y 72.019,Z 359.176,A -85,B 0,C 180,E1 -29629.971,E2 -29629.971} C_VEL
LIN {X 0,Y 75.248,Z 365.08,A -85,B 0,C 180,E1 -29639.977,E2 -29639.977} C_VEL
LIN {X 0,Y 82.628,Z 371.779,A -85,B 0,C 180,E1 -29652.049,E2 -29652.049} C_VEL
LIN {X 0,Y 63.408,Z 355.563,A -85,B 0,C 180,E1 -29666.336,E2 -29666.336} C_VEL
LIN {X 0,Y 56.496,Z 348.867,A -85,B 0,C 180,E1 -29674.18,E2 -29674.18} C_VEL
LIN {X 0,Y 47.967,Z 338.491,A -85,B 0,C 180,E1 -29689.969,E2 -29689.969} C_VEL
LIN {X 0,Y 43.378,Z 339.08,A -85,B 0,C 180,E1 -29713.565,E2 -29713.565} C_VEL
LIN {X 0,Y 43.412,Z 339.077,A -85,B 0,C 180,E1 -29729.043,E2 -29729.043} C_VEL
LIN {X 0,Y 43.702,Z 339.035,A -85,B 0,C 180,E1 -29736.478,E2 -29736.478} C_VEL
LIN {X 0,Y 43.726,Z 339.035,A -85,B 0,C 180,E1 -29739.993,E2 -29739.993} C_VEL
LIN {X 0,Y 43.792,Z 339.022,A -85,B 0,C 180,E1 -29750.063,E2 -29750.063} C_VEL
LIN {X 0,Y 43.834,Z 339.016,A -85,B 0,C 180,E1 -29761.249,E2 -29761.249} C_VEL
LIN {X 0,Y 44.22,Z 338.977,A -85,B 0,C 180,E1 -29772.437,E2 -29772.437} C_VEL
LIN {X 0,Y 44.513,Z 338.94,A -85,B 0,C 180,E1 -29780.916,E2 -29780.916} C_VEL
LIN {X 0,Y 45.096,Z 338.868,A -85,B 0,C 180,E1 -29790,E2 -29790} C_VEL
LIN {X 0,Y 44.519,Z 338.939,A -85,B 0,C 180,E1 -29799.083,E2 -29799.083} C_VEL
LIN {X 0,Y 44.165,Z 338.981,A -85,B 0,C 180,E1 -29808.558,E2 -29808.558} C_VEL
LIN {X 0,Y 43.836,Z 339.016,A -85,B 0,C 180,E1 -29818.749,E2 -29818.749} C_VEL
LIN {X 0,Y 43.813,Z 339.019,A -85,B 0,C 180,E1 -29829.915,E2 -29829.915} C_VEL
LIN {X 0,Y 43.708,Z 339.037,A -85,B 0,C 180,E1 -29839.987,E2 -29839.987} C_VEL
LIN {X 0,Y 43.659,Z 339.04,A -85,B 0,C 180,E1 -29843.599,E2 -29843.599} C_VEL
LIN {X 0,Y 43.119,Z 339.113,A -85,B 0,C 180,E1 -29850.741,E2 -29850.741} C_VEL
LIN {X 0,Y 42.428,Z 339.195,A -85,B 0,C 180,E1 -29860.666,E2 -29860.666} C_VEL
LIN {X 0,Y 44.68,Z 339.07,A -85,B 0,C 180,E1 -29883.393,E2 -29883.393} C_VEL
LIN {X 0,Y 51.758,Z 344.254,A -85,B 0,C 180,E1 -29898.1,E2 -29898.1} C_VEL
LIN {X 0,Y 53.639,Z 345.301,A -85,B 0,C 180,E1 -29900.422,E2 -29900.422} C_VEL
LIN {X 0,Y 55.868,Z 346.695,A -85,B 0,C 180,E1 -29903.786,E2 -29903.786} C_VEL
LIN {X 0,Y 57.442,Z 347.949,A -85,B 0,C 180,E1 -29907.517,E2 -29907.517} C_VEL
LIN {X 0,Y 59.047,Z 349.694,A -85,B 0,C 180,E1 -29912.43,E2 -29912.43} C_VEL
LIN {X 0,Y 60.11,Z 351.655,A -85,B 0,C 180,E1 -29915.729,E2 -29915.729} C_VEL
LIN {X 0,Y 61.075,Z 354.519,A -85,B 0,C 180,E1 -29918.216,E2 -29918.216} C_VEL
LIN {X 0,Y 64.778,Z 365.994,A -85,B 0,C 180,E1 -29924.533,E2 -29924.533} C_VEL
LIN {X 0,Y 68.227,Z 373.314,A -85,B 0,C 180,E1 -29928.759,E2 -29928.759} C_VEL
LIN {X 0,Y 67.877,Z 372.621,A -85,B 0,C 180,E1 -29931.593,E2 -29931.593} C_VEL
LIN {X 0,Y 66.079,Z 365.072,A -85,B 0,C 180,E1 -29943.127,E2 -29943.127} C_VEL
LIN {X 0,Y 66.305,Z 361.136,A -85,B 0,C 180,E1 -29948.224,E2 -29948.224} C_VEL
LIN {X 0,Y 67.451,Z 352.502,A -85,B 0,C 180,E1 -29956.534,E2 -29956.534} C_VEL
LIN {X 0,Y 66.883,Z 352.017,A -85,B 0,C 180,E1 -29957.868,E2 -29957.868} C_VEL
LIN {X 0,Y 66.16,Z 350.356,A -85,B 0,C 180,E1 -29963.902,E2 -29963.902} C_VEL
LIN {X 0,Y 66.665,Z 348.782,A -85,B 0,C 180,E1 -29970,E2 -29970} C_VEL
LIN {X 0,Y 66.652,Z 347.082,A -85,B 0,C 180,E1 -29975.483,E2 -29975.483} C_VEL
LIN {X 0,Y 65.308,Z 352.321,A -85,B 0,C 180,E1 -29985.604,E2 -29985.604} C_VEL
LIN {X 0,Y 69.1,Z 360.527,A -85,B 0,C 180,E1 -30000.567,E2 -30000.567} C_VEL
LIN {X 0,Y 72.68,Z 364.24,A -85,B 0,C 180,E1 -30007.617,E2 -30007.617} C_VEL
LIN {X 0,Y 74.083,Z 365.387,A -85,B 0,C 180,E1 -30010.62,E2 -30010.62} C_VEL
LIN {X 0,Y 57.867,Z 352.412,A -85,B 0,C 180,E1 -30022.598,E2 -30022.598} C_VEL
LIN {X 0,Y 43.831,Z 339.02,A -85,B 0,C 180,E1 -30041.283,E2 -30041.283} C_VEL
LIN {X 0,Y 37.617,Z 339.791,A -85,B 0,C 180,E1 -30059.986,E2 -30059.986} C_VEL
LIN {X 0,Y 36.267,Z 339.963,A -85,B 0,C 180,E1 -30074.322,E2 -30074.322} C_VEL
LIN {X 0,Y 36.054,Z 339.989,A -85,B 0,C 180,E1 -30082.93,E2 -30082.93} C_VEL
LIN {X 0,Y 36.526,Z 339.925,A -85,B 0,C 180,E1 -30095.238,E2 -30095.238} C_VEL
LIN {X 0,Y 36.671,Z 339.913,A -85,B 0,C 180,E1 -30099.949,E2 -30099.949} C_VEL
LIN {X 0,Y 36.71,Z 339.903,A -85,B 0,C 180,E1 -30109.953,E2 -30109.953} C_VEL
LIN {X 0,Y 36.714,Z 339.91,A -85,B 0,C 180,E1 -30114.951,E2 -30114.951} C_VEL
LIN {X 0,Y 37.046,Z 339.866,A -85,B 0,C 180,E1 -30131.493,E2 -30131.493} C_VEL
LIN {X 0,Y 37.313,Z 339.83,A -85,B 0,C 180,E1 -30139.143,E2 -30139.143} C_VEL
LIN {X 0,Y 37.959,Z 339.757,A -85,B 0,C 180,E1 -30150,E2 -30150} C_VEL
LIN {X 0,Y 37.319,Z 339.829,A -85,B 0,C 180,E1 -30160.855,E2 -30160.855} C_VEL
LIN {X 0,Y 37.059,Z 339.864,A -85,B 0,C 180,E1 -30168.565,E2 -30168.565} C_VEL
LIN {X 0,Y 36.72,Z 339.909,A -85,B 0,C 180,E1 -30185.042,E2 -30185.042} C_VEL
LIN {X 0,Y 36.724,Z 339.902,A -85,B 0,C 180,E1 -30190.071,E2 -30190.071} C_VEL
LIN {X 0,Y 36.667,Z 339.913,A -85,B 0,C 180,E1 -30200.058,E2 -30200.058} C_VEL
LIN {X 0,Y 36.425,Z 339.938,A -85,B 0,C 180,E1 -30204.65,E2 -30204.65} C_VEL
LIN {X 0,Y 35.498,Z 340.057,A -85,B 0,C 180,E1 -30216.69,E2 -30216.69} C_VEL
LIN {X 0,Y 39.446,Z 339.567,A -85,B 0,C 180,E1 -30250.925,E2 -30250.925} C_VEL
LIN {X 0,Y 48.43,Z 344.746,A -85,B 0,C 180,E1 -30265.819,E2 -30265.819} C_VEL
LIN {X 0,Y 54.343,Z 347.599,A -85,B 0,C 180,E1 -30271.163,E2 -30271.163} C_VEL
LIN {X 0,Y 60.091,Z 350.375,A -85,B 0,C 180,E1 -30276.056,E2 -30276.056} C_VEL
LIN {X 0,Y 61.075,Z 354.519,A -85,B 0,C 180,E1 -30278.216,E2 -30278.216} C_VEL
LIN {X 0,Y 61.352,Z 356.439,A -85,B 0,C 180,E1 -30280.192,E2 -30280.192} C_VEL
LIN {X 0,Y 61.65,Z 359.566,A -85,B 0,C 180,E1 -30287.707,E2 -30287.707} C_VEL
LIN {X 0,Y 62.222,Z 360.977,A -85,B 0,C 180,E1 -30289.025,E2 -30289.025} C_VEL
LIN {X 0,Y 63.603,Z 364.051,A -85,B 0,C 180,E1 -30290.68,E2 -30290.68} C_VEL
LIN {X 0,Y 63.233,Z 362.255,A -85,B 0,C 180,E1 -30296.24,E2 -30296.24} C_VEL
LIN {X 0,Y 62.861,Z 356.347,A -85,B 0,C 180,E1 -30304.675,E2 -30304.675} C_VEL
LIN {X 0,Y 63.031,Z 352.086,A -85,B 0,C 180,E1 -30309.052,E2 -30309.052} C_VEL
LIN {X 0,Y 62.27,Z 351.652,A -85,B 0,C 180,E1 -30310.209,E2 -30310.209} C_VEL
LIN {X 0,Y 60.262,Z 349.949,A -85,B 0,C 180,E1 -30316.511,E2 -30316.511} C_VEL
LIN {X 0,Y 59.435,Z 348.296,A -85,B 0,C 180,E1 -30323.209,E2 -30323.209} C_VEL
LIN {X 0,Y 59.83,Z 346.761,A -85,B 0,C 180,E1 -30330,E2 -30330} C_VEL
LIN {X 0,Y 60.026,Z 344.567,A -85,B 0,C 180,E1 -30337.759,E2 -30337.759} C_VEL
LIN {X 0,Y 59.58,Z 349.973,A -85,B 0,C 180,E1 -30349.297,E2 -30349.297} C_VEL
LIN {X 0,Y 63.856,Z 357.053,A -85,B 0,C 180,E1 -30363.388,E2 -30363.388} C_VEL
LIN {X 0,Y 65.017,Z 358.244,A -85,B 0,C 180,E1 -30365.786,E2 -30365.786} C_VEL
LIN {X 0,Y 65.862,Z 359.115,A -85,B 0,C 180,E1 -30368.646,E2 -30368.646} C_VEL
LIN {X 0,Y 52.613,Z 349.087,A -85,B 0,C 180,E1 -30378.082,E2 -30378.082} C_VEL
LIN {X 0,Y 41.156,Z 339.358,A -85,B 0,C 180,E1 -30390.843,E2 -30390.843} C_VEL
LIN {X 0,Y 32.939,Z 340.353,A -85,B 0,C 180,E1 -30407.664,E2 -30407.664} C_VEL
LIN {X 0,Y 29.129,Z 340.707,A -85,B 0,C 180,E1 -30435.185,E2 -30435.185} C_VEL
LIN {X 0,Y 29.019,Z 340.718,A -85,B 0,C 180,E1 -30448.951,E2 -30448.951} C_VEL
LIN {X 0,Y 29.521,Z 340.67,A -85,B 0,C 180,E1 -30465.551,E2 -30465.551} C_VEL
LIN {X 0,Y 29.486,Z 340.673,A -85,B 0,C 180,E1 -30481.53,E2 -30481.53} C_VEL
LIN {X 0,Y 29.854,Z 340.639,A -85,B 0,C 180,E1 -30490.274,E2 -30490.274} C_VEL
LIN {X 0,Y 30.094,Z 340.615,A -85,B 0,C 180,E1 -30496.494,E2 -30496.494} C_VEL
LIN {X 0,Y 30.781,Z 340.554,A -85,B 0,C 180,E1 -30510,E2 -30510} C_VEL
LIN {X 0,Y 30.102,Z 340.614,A -85,B 0,C 180,E1 -30523.502,E2 -30523.502} C_VEL
LIN {X 0,Y 29.864,Z 340.637,A -85,B 0,C 180,E1 -30529.777,E2 -30529.777} C_VEL
LIN {X 0,Y 29.493,Z 340.672,A -85,B 0,C 180,E1 -30538.463,E2 -30538.463} C_VEL
LIN {X 0,Y 29.519,Z 340.67,A -85,B 0,C 180,E1 -30555.582,E2 -30555.582} C_VEL
LIN {X 0,Y 28.646,Z 340.752,A -85,B 0,C 180,E1 -30570.636,E2 -30570.636} C_VEL
LIN {X 0,Y 28.434,Z 340.772,A -85,B 0,C 180,E1 -30591.368,E2 -30591.368} C_VEL
LIN {X 0,Y 35.659,Z 340.179,A -85,B 0,C 180,E1 -30621.703,E2 -30621.703} C_VEL
LIN {X 0,Y 44.773,Z 344.63,A -85,B 0,C 180,E1 -30633.339,E2 -30633.339} C_VEL
LIN {X 0,Y 51.157,Z 347.419,A -85,B 0,C 180,E1 -30638.198,E2 -30638.198} C_VEL
LIN {X 0,Y 58.643,Z 350.726,A -85,B 0,C 180,E1 -30643.571,E2 -30643.571} C_VEL
LIN {X 0,Y 62.222,Z 360.977,A -85,B 0,C 180,E1 -30649.025,E2 -30649.025} C_VEL
LIN {X 0,Y 62.331,Z 361.239,A -85,B 0,C 180,E1 -30650.03,E2 -30650.03} C_VEL
LIN {X 0,Y 61.833,Z 359.848,A -85,B 0,C 180,E1 -30652.14,E2 -30652.14} C_VEL
LIN {X 0,Y 60.172,Z 354.514,A -85,B 0,C 180,E1 -30656.472,E2 -30656.472} C_VEL
LIN {X 0,Y 60.076,Z 353.971,A -85,B 0,C 180,E1 -30657.19,E2 -30657.19} C_VEL
LIN {X 0,Y 59.846,Z 351.592,A -85,B 0,C 180,E1 -30660.608,E2 -30660.608} C_VEL
LIN {X 0,Y 53.688,Z 347.865,A -85,B 0,C 180,E1 -30674.823,E2 -30674.823} C_VEL
LIN {X 0,Y 52.975,Z 344.718,A -85,B 0,C 180,E1 -30690,E2 -30690} C_VEL
LIN {X 0,Y 53.524,Z 342.179,A -85,B 0,C 180,E1 -30700.88,E2 -30700.88} C_VEL
LIN {X 0,Y 53.996,Z 347.267,A -85,B 0,C 180,E1 -30712.984,E2 -30712.984} C_VEL
LIN {X 0,Y 57.653,Z 352.479,A -85,B 0,C 180,E1 -30724.239,E2 -30724.239} C_VEL
LIN {X 0,Y 57.516,Z 352.616,A -85,B 0,C 180,E1 -30726.234,E2 -30726.234} C_VEL
LIN {X 0,Y 47.751,Z 345.599,A -85,B 0,C 180,E1 -30732.601,E2 -30732.601} C_VEL
LIN {X 0,Y 39.707,Z 339.527,A -85,B 0,C 180,E1 -30739.657,E2 -30739.657} C_VEL
LIN {X 0,Y 30.295,Z 340.597,A -85,B 0,C 180,E1 -30752.337,E2 -30752.337} C_VEL
LIN {X 0,Y 22.979,Z 341.06,A -85,B 0,C 180,E1 -30779.977,E2 -30779.977} C_VEL
LIN {X 0,Y 21.831,Z 341.096,A -85,B 0,C 180,E1 -30798.754,E2 -30798.754} C_VEL
LIN {X 0,Y 22,Z 341.091,A -85,B 0,C 180,E1 -30819.678,E2 -30819.678} C_VEL
LIN {X 0,Y 22.18,Z 341.085,A -85,B 0,C 180,E1 -30830.675,E2 -30830.675} C_VEL
LIN {X 0,Y 22.802,Z 341.066,A -85,B 0,C 180,E1 -30852.048,E2 -30852.048} C_VEL
LIN {X 0,Y 23.557,Z 341.042,A -85,B 0,C 180,E1 -30870,E2 -30870} C_VEL
LIN {X 0,Y 22.815,Z 341.065,A -85,B 0,C 180,E1 -30887.941,E2 -30887.941} C_VEL
LIN {X 0,Y 22.184,Z 341.085,A -85,B 0,C 180,E1 -30909.318,E2 -30909.318} C_VEL
LIN {X 0,Y 21.858,Z 341.095,A -85,B 0,C 180,E1 -30920.01,E2 -30920.01} C_VEL
LIN {X 0,Y 21.078,Z 341.119,A -85,B 0,C 180,E1 -30940.55,E2 -30940.55} C_VEL
LIN {X 0,Y 29.522,Z 340.671,A -85,B 0,C 180,E1 -30988.452,E2 -30988.452} C_VEL
LIN {X 0,Y 32.737,Z 340.457,A -85,B 0,C 180,E1 -30993.355,E2 -30993.355} C_VEL
LIN {X 0,Y 48.821,Z 347.227,A -85,B 0,C 180,E1 -31006.05,E2 -31006.05} C_VEL
LIN {X 0,Y 58.461,Z 351.137,A -85,B 0,C 180,E1 -31011.445,E2 -31011.445} C_VEL
LIN {X 0,Y 60.107,Z 355.216,A -85,B 0,C 180,E1 -31013.474,E2 -31013.474} C_VEL
LIN {X 0,Y 60.379,Z 355.668,A -85,B 0,C 180,E1 -31014.581,E2 -31014.581} C_VEL
LIN {X 0,Y 60.076,Z 353.971,A -85,B 0,C 180,E1 -31017.19,E2 -31017.19} C_VEL
LIN {X 0,Y 59.081,Z 352.285,A -85,B 0,C 180,E1 -31019.593,E2 -31019.593} C_VEL
LIN {X 0,Y 56.164,Z 350.219,A -85,B 0,C 180,E1 -31022.483,E2 -31022.483} C_VEL
LIN {X 0,Y 48.99,Z 346.86,A -85,B 0,C 180,E1 -31028.854,E2 -31028.854} C_VEL
LIN {X 0,Y 47.101,Z 345.717,A -85,B 0,C 180,E1 -31033.106,E2 -31033.106} C_VEL
LIN {X 0,Y 46.135,Z 342.706,A -85,B 0,C 180,E1 -31050,E2 -31050} C_VEL
LIN {X 0,Y 47.247,Z 339.684,A -85,B 0,C 180,E1 -31064.538,E2 -31064.538} C_VEL
LIN {X 0,Y 49.973,Z 346.434,A -85,B 0,C 180,E1 -31082.436,E2 -31082.436} C_VEL
LIN {X 0,Y 39.702,Z 339.528,A -85,B 0,C 180,E1 -31088.21,E2 -31088.21} C_VEL
LIN {X 0,Y 29.036,Z 340.715,A -85,B 0,C 180,E1 -31096.563,E2 -31096.563} C_VEL
LIN {X 0,Y 15.541,Z 341.178,A -85,B 0,C 180,E1 -31139.966,E2 -31139.966} C_VEL
LIN {X 0,Y 14.72,Z 341.178,A -85,B 0,C 180,E1 -31157.275,E2 -31157.275} C_VEL
LIN {X 0,Y 14.451,Z 341.178,A -85,B 0,C 180,E1 -31169.059,E2 -31169.059} C_VEL
LIN {X 0,Y 15.057,Z 341.178,A -85,B 0,C 180,E1 -31202.175,E2 -31202.175} C_VEL
LIN {X 0,Y 15.247,Z 341.178,A -85,B 0,C 180,E1 -31207.109,E2 -31207.109} C_VEL
LIN {X 0,Y 16.232,Z 341.178,A -85,B 0,C 180,E1 -31230,E2 -31230} C_VEL
LIN {X 0,Y 15.271,Z 341.178,A -85,B 0,C 180,E1 -31253.097,E2 -31253.097} C_VEL
LIN {X 0,Y 15.09,Z 341.178,A -85,B 0,C 180,E1 -31257.758,E2 -31257.758} C_VEL
LIN {X 0,Y 14.015,Z 341.178,A -85,B 0,C 180,E1 -31289.947,E2 -31289.947} C_VEL
LIN {X 0,Y 14.595,Z 341.178,A -85,B 0,C 180,E1 -31320.036,E2 -31320.036} C_VEL
LIN {X 0,Y 23.305,Z 341.05,A -85,B 0,C 180,E1 -31357.122,E2 -31357.122} C_VEL
LIN {X 0,Y 31.338,Z 340.703,A -85,B 0,C 180,E1 -31366.567,E2 -31366.567} C_VEL
LIN {X 0,Y 43.957,Z 345.584,A -85,B 0,C 180,E1 -31373.094,E2 -31373.094} C_VEL
LIN {X 0,Y 50.83,Z 348.206,A -85,B 0,C 180,E1 -31376.075,E2 -31376.075} C_VEL
LIN {X 0,Y 53.221,Z 349.103,A -85,B 0,C 180,E1 -31378.115,E2 -31378.115} C_VEL
LIN {X 0,Y 47.101,Z 345.717,A -85,B 0,C 180,E1 -31393.106,E2 -31393.106} C_VEL
LIN {X 0,Y 45.978,Z 344.809,A -85,B 0,C 180,E1 -31397.623,E2 -31397.623} C_VEL
LIN {X 0,Y 43.109,Z 342.846,A -85,B 0,C 180,E1 -31406.806,E2 -31406.806} C_VEL
LIN {X 0,Y 40.057,Z 340.275,A -85,B 0,C 180,E1 -31422.427,E2 -31422.427} C_VEL
LIN {X 0,Y 40.575,Z 339.484,A -85,B 0,C 180,E1 -31430.757,E2 -31430.757} C_VEL
LIN {X 0,Y 41.205,Z 339.339,A -85,B 0,C 180,E1 -31433.375,E2 -31433.375} C_VEL
LIN {X 0,Y 42.027,Z 339.374,A -85,B 0,C 180,E1 -31436.005,E2 -31436.005} C_VEL
LIN {X 0,Y 41.373,Z 339.307,A -85,B 0,C 180,E1 -31437.253,E2 -31437.253} C_VEL
LIN {X 0,Y 25.347,Z 340.987,A -85,B 0,C 180,E1 -31443.679,E2 -31443.679} C_VEL
LIN {X 0,Y 8.061,Z 341.178,A -85,B 0,C 180,E1 -31499.935,E2 -31499.935} C_VEL
LIN {X 0,Y 7.446,Z 341.178,A -85,B 0,C 180,E1 -31519.296,E2 -31519.296} C_VEL
LIN {X 0,Y 7.689,Z 341.178,A -85,B 0,C 180,E1 -31565.894,E2 -31565.894} C_VEL
LIN {X 0,Y 8.666,Z 341.178,A -85,B 0,C 180,E1 -31590,E2 -31590} C_VEL
LIN {X 0,Y 7.639,Z 341.178,A -85,B 0,C 180,E1 -31613.247,E2 -31613.247} C_VEL
LIN {X 0,Y 7.164,Z 341.178,A -85,B 0,C 180,E1 -31680.073,E2 -31680.073} C_VEL
LIN {X 0,Y 25.021,Z 340.997,A -85,B 0,C 180,E1 -31737.459,E2 -31737.459} C_VEL
LIN {X 0,Y 31.202,Z 340.681,A -85,B 0,C 180,E1 -31740.03,E2 -31740.03} C_VEL
LIN {X 0,Y 41.516,Z 344.497,A -85,B 0,C 180,E1 -31742.098,E2 -31742.098} C_VEL
LIN {X 0,Y 41.611,Z 344.301,A -85,B 0,C 180,E1 -31746.747,E2 -31746.747} C_VEL
LIN {X 0,Y 39.293,Z 340.697,A -85,B 0,C 180,E1 -31770,E2 -31770} C_VEL
LIN {X 0,Y 39.312,Z 339.585,A -85,B 0,C 180,E1 -31776.415,E2 -31776.415} C_VEL
LIN {X 0,Y 41.205,Z 339.339,A -85,B 0,C 180,E1 -31793.375,E2 -31793.375} C_VEL
LIN {X 0,Y 39.887,Z 339.508,A -85,B 0,C 180,E1 -31792.928,E2 -31792.928} C_VEL
LIN {X 0,Y 35.777,Z 340.024,A -85,B 0,C 180,E1 -31785.448,E2 -31785.448} C_VEL
LIN {X 0,Y 32.37,Z 340.406,A -85,B 0,C 180,E1 -31769.739,E2 -31769.739} C_VEL
LIN {X 0,Y 32.22,Z 340.399,A -85,B 0,C 180,E1 -31762.716,E2 -31762.716} C_VEL
LIN {X 0,Y 32.803,Z 340.398,A -85,B 0,C 180,E1 -31755.744,E2 -31755.744} C_VEL
LIN {X 0,Y 32.709,Z 340.607,A -85,B 0,C 180,E1 -31752.829,E2 -31752.829} C_VEL
LIN {X 0,Y 29.355,Z 340.686,A -85,B 0,C 180,E1 -31753.324,E2 -31753.324} C_VEL
LIN {X 0,Y 14.572,Z 341.178,A -85,B 0,C 180,E1 -31754.841,E2 -31754.841} C_VEL
LIN {X 0,Y 1.681,Z 341.178,A -85,B 0,C 180,E1 -31770,E2 -31770} C_VEL
LIN {X 0,Y 7.561,Z 341.178,A -85,B 0,C 180,E1 -31791.449,E2 -31791.449} C_VEL
LIN {X 0,Y 23.313,Z 341.05,A -85,B 0,C 180,E1 -31787.545,E2 -31787.545} C_VEL
LIN {X 0,Y 31.34,Z 340.502,A -85,B 0,C 180,E1 -31787.228,E2 -31787.228} C_VEL
LIN {X 0,Y 32.517,Z 340.386,A -85,B 0,C 180,E1 -31782.482,E2 -31782.482} C_VEL
LIN {X 0,Y 32.197,Z 340.422,A -85,B 0,C 180,E1 -31770,E2 -31770} C_VEL
LIN {X 0,Y 32.22,Z 340.399,A -85,B 0,C 180,E1 -31762.716,E2 -31762.716} C_VEL
LIN {X 0,Y 32.421,Z 342.399,A -85,B 0,C 180,E1 -31759.167,E2 -31759.167} C_VEL
LIN {X 0,Y 32.421,Z 600,A -85,B 0,C 180,E1 -31759.167,E2 -31759.167} C_VEL
LIN {X 0,Y 32.421,Z 600,A -85,B 0,C 180,E1 -31759.167,E2 -31759.167}

QRS_NEXT_CUT()

QRS_NEXT()
QRS_HOME()

END
